ABB RAPID module: P106.mod

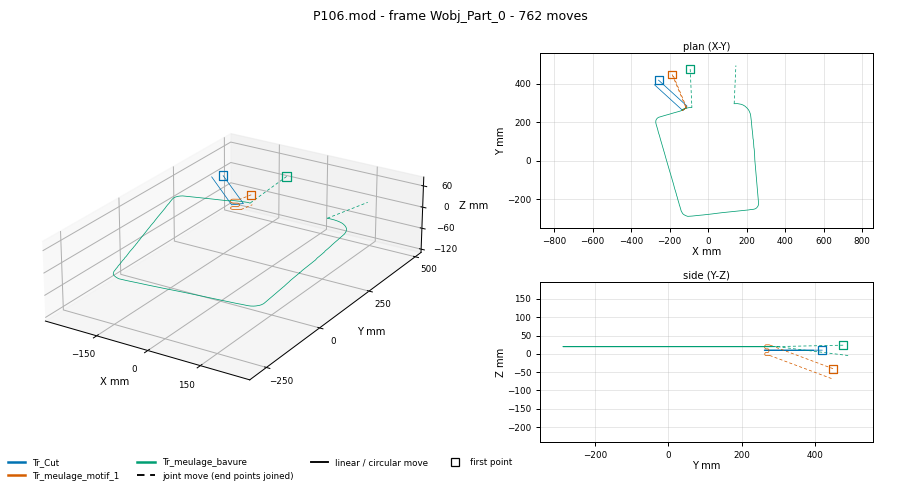
[picture p0: tool path of P106.mod in frame Wobj_Part_0, 762 of 770 moves have a stored position in this frame; points joined in program order, loops and branches not executed]
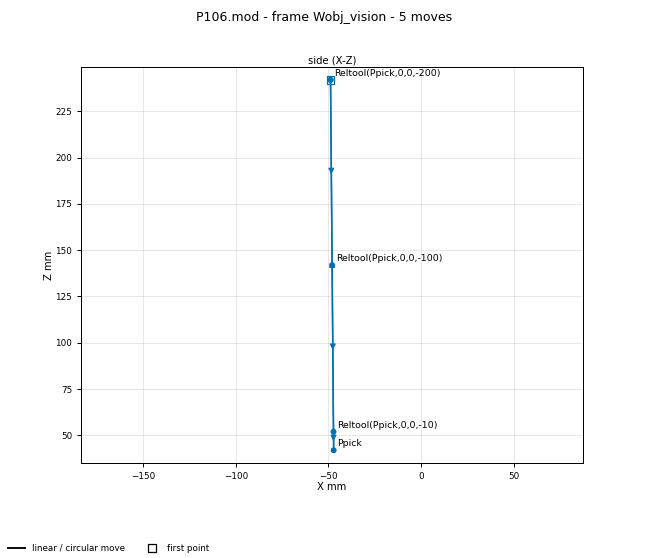
[picture p1: tool path of P106.mod in frame Wobj_vision, 5 of 770 moves have a stored position in this frame; points joined in program order, loops and branches not executed]
MODULE P106
	LOCAL CONST Speeddata vitesse_Tronconnage :=[10, 500, 0, 0];
	LOCAL CONST Robtarget Coupe_0 :=[[-123.979,269.4866875,10.1718701171875],[0.659483403277492,0.659350185940918,-0.255455147334473,-0.255111036220579],[0,0,0,0],[8.999999E+09,8.999999E+09,8.999999E+09,8.999999E+09,8.999999E+09,8.999999E+09]];
	LOCAL CONST Robtarget Tr_meulage_motif_1_App1 :=[[-187.295514074662,449.36288798166,-40.5098213895633],[0.160101054175836,-0.114155213921264,0.569221589744271,-0.798325135114373],[0,0,0,0],[8.999999E+09,8.999999E+09,8.999999E+09,8.999999E+09,8.999999E+09,8.999999E+09]];
	LOCAL CONST Robtarget Tr_meulage_motif_1_App2 :=[[-118.034451875608,283.626825649083,21.4132187938031],[0.160101054175836,-0.114155213921264,0.569221589744271,-0.798325135114373],[0,0,0,0],[8.999999E+09,8.999999E+09,8.999999E+09,8.999999E+09,8.999999E+09,8.999999E+09]];
	LOCAL CONST Robtarget Tr_meulage_motif_1_P0 :=[[-114.3891328125,274.903875,24.672326171875],[0.160101054175836,-0.114155213921264,0.569221589744271,-0.798325135114373],[0,0,0,0],[8.999999E+09,8.999999E+09,8.999999E+09,8.999999E+09,8.999999E+09,8.999999E+09]];
	LOCAL CONST Robtarget Tr_meulage_motif_1_P1 :=[[-115.2604296875,274.413125,24.672283203125],[0.160101054175836,-0.114155213921264,0.569221589744271,-0.798325135114373],[0,0,0,0],[8.999999E+09,8.999999E+09,8.999999E+09,8.999999E+09,8.999999E+09,8.999999E+09]];
	LOCAL CONST Robtarget Tr_meulage_motif_1_P2 :=[[-116.1317265625,273.922375,24.6722421875],[0.160101054175836,-0.114155213921264,0.569221589744271,-0.798325135114373],[0,0,0,0],[8.999999E+09,8.999999E+09,8.999999E+09,8.999999E+09,8.999999E+09,8.999999E+09]];
	LOCAL CONST Robtarget Tr_meulage_motif_1_P3 :=[[-117.0030234375,273.43159375,24.67219921875],[0.160101054175836,-0.114155213921264,0.569221589744271,-0.798325135114373],[0,0,0,0],[8.999999E+09,8.999999E+09,8.999999E+09,8.999999E+09,8.999999E+09,8.999999E+09]];
	LOCAL CONST Robtarget Tr_meulage_motif_1_P4 :=[[-117.8743203125,272.94084375,24.672158203125],[0.160101054175836,-0.114155213921264,0.569221589744271,-0.798325135114373],[0,0,0,0],[8.999999E+09,8.999999E+09,8.999999E+09,8.999999E+09,8.999999E+09,8.999999E+09]];
	LOCAL CONST Robtarget Tr_meulage_motif_1_P5 :=[[-118.745609375,272.45009375,24.672115234375],[0.160101054175836,-0.114155213921264,0.569221589744271,-0.798325135114373],[0,0,0,0],[8.999999E+09,8.999999E+09,8.999999E+09,8.999999E+09,8.999999E+09,8.999999E+09]];
	LOCAL CONST Robtarget Tr_meulage_motif_1_P6 :=[[-119.61690625,271.95934375,24.67207421875],[0.160101054175836,-0.114155213921264,0.569221589744271,-0.798325135114373],[0,0,0,0],[8.999999E+09,8.999999E+09,8.999999E+09,8.999999E+09,8.999999E+09,8.999999E+09]];
	LOCAL CONST Robtarget Tr_meulage_motif_1_P7 :=[[-120.488203125,271.4685625,24.67203125],[0.160101054175836,-0.114155213921264,0.569221589744271,-0.798325135114373],[0,0,0,0],[8.999999E+09,8.999999E+09,8.999999E+09,8.999999E+09,8.999999E+09,8.999999E+09]];
	LOCAL CONST Robtarget Tr_meulage_motif_1_P8 :=[[-121.3595,270.9778125,24.671990234375],[0.160101054175836,-0.114155213921264,0.569221589744271,-0.798325135114373],[0,0,0,0],[8.999999E+09,8.999999E+09,8.999999E+09,8.999999E+09,8.999999E+09,8.999999E+09]];
	LOCAL CONST Robtarget Tr_meulage_motif_1_P9 :=[[-122.230796875,270.4870625,24.671947265625],[0.160101054175836,-0.114155213921264,0.569221589744271,-0.798325135114373],[0,0,0,0],[8.999999E+09,8.999999E+09,8.999999E+09,8.999999E+09,8.999999E+09,8.999999E+09]];
	LOCAL CONST Robtarget Tr_meulage_motif_1_P10 :=[[-123.10209375,269.9963125,24.67190625],[0.160101054175836,-0.114155213921264,0.569221589744271,-0.798325135114373],[0,0,0,0],[8.999999E+09,8.999999E+09,8.999999E+09,8.999999E+09,8.999999E+09,8.999999E+09]];
	LOCAL CONST Robtarget Tr_meulage_motif_1_P11 :=[[-123.973390625,269.50553125,24.671865234375],[0.160101054175836,-0.114155213921264,0.569221589744271,-0.798325135114373],[0,0,0,0],[8.999999E+09,8.999999E+09,8.999999E+09,8.999999E+09,8.999999E+09,8.999999E+09]];
	LOCAL CONST Robtarget Tr_meulage_motif_1_P12 :=[[-124.8446796875,269.01478125,24.671822265625],[0.160101054175836,-0.114155213921264,0.569221589744271,-0.798325135114373],[0,0,0,0],[8.999999E+09,8.999999E+09,8.999999E+09,8.999999E+09,8.999999E+09,8.999999E+09]];
	LOCAL CONST Robtarget Tr_meulage_motif_1_P13 :=[[-125.7159765625,268.52403125,24.67178125],[0.160101054175836,-0.114155213921264,0.569221589744271,-0.798325135114373],[0,0,0,0],[8.999999E+09,8.999999E+09,8.999999E+09,8.999999E+09,8.999999E+09,8.999999E+09]];
	LOCAL CONST Robtarget Tr_meulage_motif_1_P14 :=[[-126.5872734375,268.03325,24.67173828125],[0.160101054175836,-0.114155213921264,0.569221589744271,-0.798325135114373],[0,0,0,0],[8.999999E+09,8.999999E+09,8.999999E+09,8.999999E+09,8.999999E+09,8.999999E+09]];
	LOCAL CONST Robtarget Tr_meulage_motif_1_P15 :=[[-127.4585703125,267.5425,24.671697265625],[0.160101054175836,-0.114155213921264,0.569221589744271,-0.798325135114373],[0,0,0,0],[8.999999E+09,8.999999E+09,8.999999E+09,8.999999E+09,8.999999E+09,8.999999E+09]];
	LOCAL CONST Robtarget Tr_meulage_motif_1_P16 :=[[-128.3298671875,267.05175,24.671654296875],[0.160101054175836,-0.114155213921264,0.569221589744271,-0.798325135114373],[0,0,0,0],[8.999999E+09,8.999999E+09,8.999999E+09,8.999999E+09,8.999999E+09,8.999999E+09]];
	LOCAL CONST Robtarget Tr_meulage_motif_1_P17 :=[[-129.2011640625,266.561,24.67161328125],[0.160101054175836,-0.114155213921264,0.569221589744271,-0.798325135114373],[0,0,0,0],[8.999999E+09,8.999999E+09,8.999999E+09,8.999999E+09,8.999999E+09,8.999999E+09]];
	LOCAL CONST Robtarget Tr_meulage_motif_1_P18 :=[[-130.072453125,266.07021875,24.6715703125],[0.160101054175836,-0.114155213921264,0.569221589744271,-0.798325135114373],[0,0,0,0],[8.999999E+09,8.999999E+09,8.999999E+09,8.999999E+09,8.999999E+09,8.999999E+09]];
	LOCAL CONST Robtarget Tr_meulage_motif_1_P19 :=[[-130.93721875,265.58303125,24.560935546875],[0.160101054175836,-0.114155213921264,0.569221589744271,-0.798325135114373],[0,0,0,0],[8.999999E+09,8.999999E+09,8.999999E+09,8.999999E+09,8.999999E+09,8.999999E+09]];
	LOCAL CONST Robtarget Tr_meulage_motif_1_P20 :=[[-131.761796875,265.118375,24.349708984375],[0.160101054175836,-0.114155213921264,0.569221589744271,-0.798325135114373],[0,0,0,0],[8.999999E+09,8.999999E+09,8.999999E+09,8.999999E+09,8.999999E+09,8.999999E+09]];
	LOCAL CONST Robtarget Tr_meulage_motif_1_P21 :=[[-132.504625,264.69965625,24.077828125],[0.160101054175836,-0.114155213921264,0.569221589744271,-0.798325135114373],[0,0,0,0],[8.999999E+09,8.999999E+09,8.999999E+09,8.999999E+09,8.999999E+09,8.999999E+09]];
	LOCAL CONST Robtarget Tr_meulage_motif_1_P22 :=[[-133.15790625,264.33140625,23.801859375],[0.160101054175836,-0.114155213921264,0.569221589744271,-0.798325135114373],[0,0,0,0],[8.999999E+09,8.999999E+09,8.999999E+09,8.999999E+09,8.999999E+09,8.999999E+09]];
	LOCAL CONST Robtarget Tr_meulage_motif_1_P23 :=[[-134.116953125,263.7905625,23.185689453125],[0.160101054175836,-0.114155213921264,0.569221589744271,-0.798325135114373],[0,0,0,0],[8.999999E+09,8.999999E+09,8.999999E+09,8.999999E+09,8.999999E+09,8.999999E+09]];
	LOCAL CONST Robtarget Tr_meulage_motif_1_P24 :=[[-135.008625,263.28740625,22.337990234375],[0.160101054175836,-0.114155213921264,0.569221589744271,-0.798325135114373],[0,0,0,0],[8.999999E+09,8.999999E+09,8.999999E+09,8.999999E+09,8.999999E+09,8.999999E+09]];
	LOCAL CONST Robtarget Tr_meulage_motif_1_P25 :=[[-135.746671875,262.87059375,21.314080078125],[0.160101054175836,-0.114155213921264,0.569221589744271,-0.798325135114373],[0,0,0,0],[8.999999E+09,8.999999E+09,8.999999E+09,8.999999E+09,8.999999E+09,8.999999E+09]];
	LOCAL CONST Robtarget Tr_meulage_motif_1_P26 :=[[-136.1714375,262.630125,20.197873046875],[0.160101054175836,-0.114155213921264,0.569221589744271,-0.798325135114373],[0,0,0,0],[8.999999E+09,8.999999E+09,8.999999E+09,8.999999E+09,8.999999E+09,8.999999E+09]];
	LOCAL CONST Robtarget Tr_meulage_motif_1_P27 :=[[-136.194671875,262.61628125,19.50190234375],[0.160101054175836,-0.114155213921264,0.569221589744271,-0.798325135114373],[0,0,0,0],[8.999999E+09,8.999999E+09,8.999999E+09,8.999999E+09,8.999999E+09,8.999999E+09]];
	LOCAL CONST Robtarget Tr_meulage_motif_1_P28 :=[[-136.19434375,262.61575,18.840654296875],[0.160101054175836,-0.114155213921264,0.569221589744271,-0.798325135114373],[0,0,0,0],[8.999999E+09,8.999999E+09,8.999999E+09,8.999999E+09,8.999999E+09,8.999999E+09]];
	LOCAL CONST Robtarget Tr_meulage_motif_1_P29 :=[[-136.146203125,262.64215625,18.1795625],[0.160101054175836,-0.114155213921264,0.569221589744271,-0.798325135114373],[0,0,0,0],[8.999999E+09,8.999999E+09,8.999999E+09,8.999999E+09,8.999999E+09,8.999999E+09]];
	LOCAL CONST Robtarget Tr_meulage_motif_1_P30 :=[[-135.7115625,262.88578125,17.077833984375],[0.160101054175836,-0.114155213921264,0.569221589744271,-0.798325135114373],[0,0,0,0],[8.999999E+09,8.999999E+09,8.999999E+09,8.999999E+09,8.999999E+09,8.999999E+09]];
	LOCAL CONST Robtarget Tr_meulage_motif_1_P31 :=[[-134.9646875,263.305375,16.0712451171875],[0.160101054175836,-0.114155213921264,0.569221589744271,-0.798325135114373],[0,0,0,0],[8.999999E+09,8.999999E+09,8.999999E+09,8.999999E+09,8.999999E+09,8.999999E+09]];
	LOCAL CONST Robtarget Tr_meulage_motif_1_P32 :=[[-134.072578125,263.8069375,15.2424130859375],[0.160101054175836,-0.114155213921264,0.569221589744271,-0.798325135114373],[0,0,0,0],[8.999999E+09,8.999999E+09,8.999999E+09,8.999999E+09,8.999999E+09,8.999999E+09]];
	LOCAL CONST Robtarget Tr_meulage_motif_1_P33 :=[[-133.47371875,264.14384375,14.8466923828125],[0.160101054175836,-0.114155213921264,0.569221589744271,-0.798325135114373],[0,0,0,0],[8.999999E+09,8.999999E+09,8.999999E+09,8.999999E+09,8.999999E+09,8.999999E+09]];
	LOCAL CONST Robtarget Tr_meulage_motif_1_P34 :=[[-132.464375,264.7118125,14.3592099609375],[0.160101054175836,-0.114155213921264,0.569221589744271,-0.798325135114373],[0,0,0,0],[8.999999E+09,8.999999E+09,8.999999E+09,8.999999E+09,8.999999E+09,8.999999E+09]];
	LOCAL CONST Robtarget Tr_meulage_motif_1_P35 :=[[-131.72796875,265.1263125,14.0951513671875],[0.160101054175836,-0.114155213921264,0.569221589744271,-0.798325135114373],[0,0,0,0],[8.999999E+09,8.999999E+09,8.999999E+09,8.999999E+09,8.999999E+09,8.999999E+09]];
	LOCAL CONST Robtarget Tr_meulage_motif_1_P36 :=[[-130.915828125,265.58353125,13.8907216796875],[0.160101054175836,-0.114155213921264,0.569221589744271,-0.798325135114373],[0,0,0,0],[8.999999E+09,8.999999E+09,8.999999E+09,8.999999E+09,8.999999E+09,8.999999E+09]];
	LOCAL CONST Robtarget Tr_meulage_motif_1_P37 :=[[-130.0605390625,266.06515625,13.782169921875],[0.160101054175836,-0.114155213921264,0.569221589744271,-0.798325135114373],[0,0,0,0],[8.999999E+09,8.999999E+09,8.999999E+09,8.999999E+09,8.999999E+09,8.999999E+09]];
	LOCAL CONST Robtarget Tr_meulage_motif_1_P38 :=[[-129.195671875,266.5521875,13.6716171875],[0.160101054175836,-0.114155213921264,0.569221589744271,-0.798325135114373],[0,0,0,0],[8.999999E+09,8.999999E+09,8.999999E+09,8.999999E+09,8.999999E+09,8.999999E+09]];
	LOCAL CONST Robtarget Tr_meulage_motif_1_P39 :=[[-128.324375,267.0429375,13.6716591796875],[0.160101054175836,-0.114155213921264,0.569221589744271,-0.798325135114373],[0,0,0,0],[8.999999E+09,8.999999E+09,8.999999E+09,8.999999E+09,8.999999E+09,8.999999E+09]];
	LOCAL CONST Robtarget Tr_meulage_motif_1_P40 :=[[-127.453078125,267.5336875,13.671701171875],[0.160101054175836,-0.114155213921264,0.569221589744271,-0.798325135114373],[0,0,0,0],[8.999999E+09,8.999999E+09,8.999999E+09,8.999999E+09,8.999999E+09,8.999999E+09]];
	LOCAL CONST Robtarget Tr_meulage_motif_1_P41 :=[[-126.58178125,268.02446875,13.6717431640625],[0.160101054175836,-0.114155213921264,0.569221589744271,-0.798325135114373],[0,0,0,0],[8.999999E+09,8.999999E+09,8.999999E+09,8.999999E+09,8.999999E+09,8.999999E+09]];
	LOCAL CONST Robtarget Tr_meulage_motif_1_P42 :=[[-125.710484375,268.51521875,13.67178515625],[0.160101054175836,-0.114155213921264,0.569221589744271,-0.798325135114373],[0,0,0,0],[8.999999E+09,8.999999E+09,8.999999E+09,8.999999E+09,8.999999E+09,8.999999E+09]];
	LOCAL CONST Robtarget Tr_meulage_motif_1_P43 :=[[-124.8391875,269.00596875,13.6718271484375],[0.160101054175836,-0.114155213921264,0.569221589744271,-0.798325135114373],[0,0,0,0],[8.999999E+09,8.999999E+09,8.999999E+09,8.999999E+09,8.999999E+09,8.999999E+09]];
	LOCAL CONST Robtarget Tr_meulage_motif_1_P44 :=[[-123.9678984375,269.49671875,13.671869140625],[0.160101054175836,-0.114155213921264,0.569221589744271,-0.798325135114373],[0,0,0,0],[8.999999E+09,8.999999E+09,8.999999E+09,8.999999E+09,8.999999E+09,8.999999E+09]];
	LOCAL CONST Robtarget Tr_meulage_motif_1_P45 :=[[-123.0966015625,269.9875,13.6719111328125],[0.160101054175836,-0.114155213921264,0.569221589744271,-0.798325135114373],[0,0,0,0],[8.999999E+09,8.999999E+09,8.999999E+09,8.999999E+09,8.999999E+09,8.999999E+09]];
	LOCAL CONST Robtarget Tr_meulage_motif_1_P46 :=[[-122.2253046875,270.47825,13.671953125],[0.160101054175836,-0.114155213921264,0.569221589744271,-0.798325135114373],[0,0,0,0],[8.999999E+09,8.999999E+09,8.999999E+09,8.999999E+09,8.999999E+09,8.999999E+09]];
	LOCAL CONST Robtarget Tr_meulage_motif_1_P47 :=[[-121.3540078125,270.969,13.6719951171875],[0.160101054175836,-0.114155213921264,0.569221589744271,-0.798325135114373],[0,0,0,0],[8.999999E+09,8.999999E+09,8.999999E+09,8.999999E+09,8.999999E+09,8.999999E+09]];
	LOCAL CONST Robtarget Tr_meulage_motif_1_P48 :=[[-120.4827109375,271.45975,13.672037109375],[0.160101054175836,-0.114155213921264,0.569221589744271,-0.798325135114373],[0,0,0,0],[8.999999E+09,8.999999E+09,8.999999E+09,8.999999E+09,8.999999E+09,8.999999E+09]];
	LOCAL CONST Robtarget Tr_meulage_motif_1_P49 :=[[-119.61784375,271.94678125,13.5614853515625],[0.160101054175836,-0.114155213921264,0.569221589744271,-0.798325135114373],[0,0,0,0],[8.999999E+09,8.999999E+09,8.999999E+09,8.999999E+09,8.999999E+09,8.999999E+09]];
	LOCAL CONST Robtarget Tr_meulage_motif_1_P50 :=[[-118.7930546875,272.411125,13.3503369140625],[0.160101054175836,-0.114155213921264,0.569221589744271,-0.798325135114373],[0,0,0,0],[8.999999E+09,8.999999E+09,8.999999E+09,8.999999E+09,8.999999E+09,8.999999E+09]];
	LOCAL CONST Robtarget Tr_meulage_motif_1_P51 :=[[-118.049953125,272.829375,13.078529296875],[0.160101054175836,-0.114155213921264,0.569221589744271,-0.798325135114373],[0,0,0,0],[8.999999E+09,8.999999E+09,8.999999E+09,8.999999E+09,8.999999E+09,8.999999E+09]];
	LOCAL CONST Robtarget Tr_meulage_motif_1_P52 :=[[-117.4298671875,273.1783125,12.7744033203125],[0.160101054175836,-0.114155213921264,0.569221589744271,-0.798325135114373],[0,0,0,0],[8.999999E+09,8.999999E+09,8.999999E+09,8.999999E+09,8.999999E+09,8.999999E+09]];
	LOCAL CONST Robtarget Tr_meulage_motif_1_P53 :=[[-116.5282109375,273.6854375,12.111916015625],[0.160101054175836,-0.114155213921264,0.569221589744271,-0.798325135114373],[0,0,0,0],[8.999999E+09,8.999999E+09,8.999999E+09,8.999999E+09,8.999999E+09,8.999999E+09]];
	LOCAL CONST Robtarget Tr_meulage_motif_1_P54 :=[[-115.74190625,274.127375,11.2100166015625],[0.160101054175836,-0.114155213921264,0.569221589744271,-0.798325135114373],[0,0,0,0],[8.999999E+09,8.999999E+09,8.999999E+09,8.999999E+09,8.999999E+09,8.999999E+09]];
	LOCAL CONST Robtarget Tr_meulage_motif_1_P55 :=[[-115.275265625,274.3890625,10.1640078125],[0.160101054175836,-0.114155213921264,0.569221589744271,-0.798325135114373],[0,0,0,0],[8.999999E+09,8.999999E+09,8.999999E+09,8.999999E+09,8.999999E+09,8.999999E+09]];
	LOCAL CONST Robtarget Tr_meulage_motif_1_P56 :=[[-115.113921875,274.4791875,9.470796875],[0.160101054175836,-0.114155213921264,0.569221589744271,-0.798325135114373],[0,0,0,0],[8.999999E+09,8.999999E+09,8.999999E+09,8.999999E+09,8.999999E+09,8.999999E+09]];
	LOCAL CONST Robtarget Tr_meulage_motif_1_P57 :=[[-115.0579140625,274.50990625,8.7007998046875],[0.160101054175836,-0.114155213921264,0.569221589744271,-0.798325135114373],[0,0,0,0],[8.999999E+09,8.999999E+09,8.999999E+09,8.999999E+09,8.999999E+09,8.999999E+09]];
	LOCAL CONST Robtarget Tr_meulage_motif_1_P58 :=[[-115.1158515625,274.4764375,7.9309228515625],[0.160101054175836,-0.114155213921264,0.569221589744271,-0.798325135114373],[0,0,0,0],[8.999999E+09,8.999999E+09,8.999999E+09,8.999999E+09,8.999999E+09,8.999999E+09]];
	LOCAL CONST Robtarget Tr_meulage_motif_1_P59 :=[[-115.480890625,274.269625,6.82265576171875],[0.160101054175836,-0.114155213921264,0.569221589744271,-0.798325135114373],[0,0,0,0],[8.999999E+09,8.999999E+09,8.999999E+09,8.999999E+09,8.999999E+09,8.999999E+09]];
	LOCAL CONST Robtarget Tr_meulage_motif_1_P60 :=[[-115.8415859375,274.06584375,6.236951171875],[0.160101054175836,-0.114155213921264,0.569221589744271,-0.798325135114373],[0,0,0,0],[8.999999E+09,8.999999E+09,8.999999E+09,8.999999E+09,8.999999E+09,8.999999E+09]];
	LOCAL CONST Robtarget Tr_meulage_motif_1_P61 :=[[-116.6140859375,273.62975,5.3497890625],[0.160101054175836,-0.114155213921264,0.569221589744271,-0.798325135114373],[0,0,0,0],[8.999999E+09,8.999999E+09,8.999999E+09,8.999999E+09,8.999999E+09,8.999999E+09]];
	LOCAL CONST Robtarget Tr_meulage_motif_1_P62 :=[[-117.1241875,273.342,4.9354521484375],[0.160101054175836,-0.114155213921264,0.569221589744271,-0.798325135114373],[0,0,0,0],[8.999999E+09,8.999999E+09,8.999999E+09,8.999999E+09,8.999999E+09,8.999999E+09]];
	LOCAL CONST Robtarget Tr_meulage_motif_1_P63 :=[[-118.0979453125,272.7929375,4.39131201171875],[0.160101054175836,-0.114155213921264,0.569221589744271,-0.798325135114373],[0,0,0,0],[8.999999E+09,8.999999E+09,8.999999E+09,8.999999E+09,8.999999E+09,8.999999E+09]];
	LOCAL CONST Robtarget Tr_meulage_motif_1_P64 :=[[-118.8171328125,272.38753125,4.09577734375],[0.160101054175836,-0.114155213921264,0.569221589744271,-0.798325135114373],[0,0,0,0],[8.999999E+09,8.999999E+09,8.999999E+09,8.999999E+09,8.999999E+09,8.999999E+09]];
	LOCAL CONST Robtarget Tr_meulage_motif_1_P65 :=[[-119.629078125,271.93,3.89126977539062],[0.160101054175836,-0.114155213921264,0.569221589744271,-0.798325135114373],[0,0,0,0],[8.999999E+09,8.999999E+09,8.999999E+09,8.999999E+09,8.999999E+09,8.999999E+09]];
	LOCAL CONST Robtarget Tr_meulage_motif_1_P66 :=[[-120.4842578125,271.4481875,3.782634765625],[0.160101054175836,-0.114155213921264,0.569221589744271,-0.798325135114373],[0,0,0,0],[8.999999E+09,8.999999E+09,8.999999E+09,8.999999E+09,8.999999E+09,8.999999E+09]];
	LOCAL CONST Robtarget Tr_meulage_motif_1_P67 :=[[-121.349015625,270.961,3.67199951171875],[0.160101054175836,-0.114155213921264,0.569221589744271,-0.798325135114373],[0,0,0,0],[8.999999E+09,8.999999E+09,8.999999E+09,8.999999E+09,8.999999E+09,8.999999E+09]];
	LOCAL CONST Robtarget Tr_meulage_motif_1_P68 :=[[-122.2203125,270.47025,3.67195751953125],[0.160101054175836,-0.114155213921264,0.569221589744271,-0.798325135114373],[0,0,0,0],[8.999999E+09,8.999999E+09,8.999999E+09,8.999999E+09,8.999999E+09,8.999999E+09]];
	LOCAL CONST Robtarget Tr_meulage_motif_1_P69 :=[[-123.091609375,269.97946875,3.67191552734375],[0.160101054175836,-0.114155213921264,0.569221589744271,-0.798325135114373],[0,0,0,0],[8.999999E+09,8.999999E+09,8.999999E+09,8.999999E+09,8.999999E+09,8.999999E+09]];
	LOCAL CONST Robtarget Tr_meulage_motif_1_P70 :=[[-123.96290625,269.48871875,3.67187353515625],[0.160101054175836,-0.114155213921264,0.569221589744271,-0.798325135114373],[0,0,0,0],[8.999999E+09,8.999999E+09,8.999999E+09,8.999999E+09,8.999999E+09,8.999999E+09]];
	LOCAL CONST Robtarget Tr_meulage_motif_1_P71 :=[[-124.8341953125,268.99796875,3.67183178710938],[0.160101054175836,-0.114155213921264,0.569221589744271,-0.798325135114373],[0,0,0,0],[8.999999E+09,8.999999E+09,8.999999E+09,8.999999E+09,8.999999E+09,8.999999E+09]];
	LOCAL CONST Robtarget Tr_meulage_motif_1_P72 :=[[-125.7054921875,268.50721875,3.67178979492187],[0.160101054175836,-0.114155213921264,0.569221589744271,-0.798325135114373],[0,0,0,0],[8.999999E+09,8.999999E+09,8.999999E+09,8.999999E+09,8.999999E+09,8.999999E+09]];
	LOCAL CONST Robtarget Tr_meulage_motif_1_P73 :=[[-126.5767890625,268.0164375,3.67174780273438],[0.160101054175836,-0.114155213921264,0.569221589744271,-0.798325135114373],[0,0,0,0],[8.999999E+09,8.999999E+09,8.999999E+09,8.999999E+09,8.999999E+09,8.999999E+09]];
	LOCAL CONST Robtarget Tr_meulage_motif_1_P74 :=[[-127.4480859375,267.5256875,3.67170581054688],[0.160101054175836,-0.114155213921264,0.569221589744271,-0.798325135114373],[0,0,0,0],[8.999999E+09,8.999999E+09,8.999999E+09,8.999999E+09,8.999999E+09,8.999999E+09]];
	LOCAL CONST Robtarget Tr_meulage_motif_1_P75 :=[[-128.3193828125,267.0349375,3.67166381835938],[0.160101054175836,-0.114155213921264,0.569221589744271,-0.798325135114373],[0,0,0,0],[8.999999E+09,8.999999E+09,8.999999E+09,8.999999E+09,8.999999E+09,8.999999E+09]];
	LOCAL CONST Robtarget Tr_meulage_motif_1_P76 :=[[-129.1906796875,266.54415625,3.67162182617187],[0.160101054175836,-0.114155213921264,0.569221589744271,-0.798325135114373],[0,0,0,0],[8.999999E+09,8.999999E+09,8.999999E+09,8.999999E+09,8.999999E+09,8.999999E+09]];
	LOCAL CONST Robtarget Tr_meulage_motif_1_P77 :=[[-130.0619765625,266.05340625,3.671580078125],[0.160101054175836,-0.114155213921264,0.569221589744271,-0.798325135114373],[0,0,0,0],[8.999999E+09,8.999999E+09,8.999999E+09,8.999999E+09,8.999999E+09,8.999999E+09]];
	LOCAL CONST Robtarget Tr_meulage_motif_1_P78 :=[[-130.926734375,265.56621875,3.56094458007813],[0.160101054175836,-0.114155213921264,0.569221589744271,-0.798325135114373],[0,0,0,0],[8.999999E+09,8.999999E+09,8.999999E+09,8.999999E+09,8.999999E+09,8.999999E+09]];
	LOCAL CONST Robtarget Tr_meulage_motif_1_P79 :=[[-131.7513125,265.10153125,3.34971752929688],[0.160101054175836,-0.114155213921264,0.569221589744271,-0.798325135114373],[0,0,0,0],[8.999999E+09,8.999999E+09,8.999999E+09,8.999999E+09,8.999999E+09,8.999999E+09]];
	LOCAL CONST Robtarget Tr_meulage_motif_1_P80 :=[[-132.494140625,264.68284375,3.07783813476563],[0.160101054175836,-0.114155213921264,0.569221589744271,-0.798325135114373],[0,0,0,0],[8.999999E+09,8.999999E+09,8.999999E+09,8.999999E+09,8.999999E+09,8.999999E+09]];
	LOCAL CONST Robtarget Tr_meulage_motif_1_P81 :=[[-133.147421875,264.31459375,2.80186938476563],[0.160101054175836,-0.114155213921264,0.569221589744271,-0.798325135114373],[0,0,0,0],[8.999999E+09,8.999999E+09,8.999999E+09,8.999999E+09,8.999999E+09,8.999999E+09]];
	LOCAL CONST Robtarget Tr_meulage_motif_1_P82 :=[[-134.10646875,263.77375,2.18569848632813],[0.160101054175836,-0.114155213921264,0.569221589744271,-0.798325135114373],[0,0,0,0],[8.999999E+09,8.999999E+09,8.999999E+09,8.999999E+09,8.999999E+09,8.999999E+09]];
	LOCAL CONST Robtarget Tr_meulage_motif_1_P83 :=[[-134.939609375,263.3035,1.29168994140625],[0.160101054175836,-0.114155213921264,0.569221589744271,-0.798325135114373],[0,0,0,0],[8.999999E+09,8.999999E+09,8.999999E+09,8.999999E+09,8.999999E+09,8.999999E+09]];
	LOCAL CONST Robtarget Tr_meulage_motif_1_P84 :=[[-135.469796875,263.0036875,0.205664825439453],[0.160101054175836,-0.114155213921264,0.569221589744271,-0.798325135114373],[0,0,0,0],[8.999999E+09,8.999999E+09,8.999999E+09,8.999999E+09,8.999999E+09,8.999999E+09]];
	LOCAL CONST Robtarget Tr_meulage_motif_1_P85 :=[[-135.616828125,262.9198125,-0.778716857910156],[0.160101054175836,-0.114155213921264,0.569221589744271,-0.798325135114373],[0,0,0,0],[8.999999E+09,8.999999E+09,8.999999E+09,8.999999E+09,8.999999E+09,8.999999E+09]];
	LOCAL CONST Robtarget Tr_meulage_motif_1_P86 :=[[-135.502171875,262.9841875,-0.983367492675781],[0.160101054175836,-0.114155213921264,0.569221589744271,-0.798325135114373],[0,0,0,0],[8.999999E+09,8.999999E+09,8.999999E+09,8.999999E+09,8.999999E+09,8.999999E+09]];
	LOCAL CONST Robtarget Tr_meulage_motif_1_P87 :=[[-135.3943125,263.04415625,-1.70976818847656],[0.160101054175836,-0.114155213921264,0.569221589744271,-0.798325135114373],[0,0,0,0],[8.999999E+09,8.999999E+09,8.999999E+09,8.999999E+09,8.999999E+09,8.999999E+09]];
	LOCAL CONST Robtarget Tr_meulage_motif_1_P88 :=[[-134.797875,263.3790625,-2.64664526367187],[0.160101054175836,-0.114155213921264,0.569221589744271,-0.798325135114373],[0,0,0,0],[8.999999E+09,8.999999E+09,8.999999E+09,8.999999E+09,8.999999E+09,8.999999E+09]];
	LOCAL CONST Robtarget Tr_meulage_motif_1_P89 :=[[-134.311796875,263.65234375,-3.11043432617187],[0.160101054175836,-0.114155213921264,0.569221589744271,-0.798325135114373],[0,0,0,0],[8.999999E+09,8.999999E+09,8.999999E+09,8.999999E+09,8.999999E+09,8.999999E+09]];
	LOCAL CONST Robtarget Tr_meulage_motif_1_P90 :=[[-133.3266875,264.20665625,-3.64082421875],[0.160101054175836,-0.114155213921264,0.569221589744271,-0.798325135114373],[0,0,0,0],[8.999999E+09,8.999999E+09,8.999999E+09,8.999999E+09,8.999999E+09,8.999999E+09]];
	LOCAL CONST Robtarget Tr_meulage_motif_1_P91 :=[[-132.59028125,264.621125,-3.90488232421875],[0.160101054175836,-0.114155213921264,0.569221589744271,-0.798325135114373],[0,0,0,0],[8.999999E+09,8.999999E+09,8.999999E+09,8.999999E+09,8.999999E+09,8.999999E+09]];
	LOCAL CONST Robtarget Tr_meulage_motif_1_P92 :=[[-131.778140625,265.078375,-4.10931201171875],[0.160101054175836,-0.114155213921264,0.569221589744271,-0.798325135114373],[0,0,0,0],[8.999999E+09,8.999999E+09,8.999999E+09,8.999999E+09,8.999999E+09,8.999999E+09]];
	LOCAL CONST Robtarget Tr_meulage_motif_1_P93 :=[[-130.9228515625,265.56,-4.2178642578125],[0.160101054175836,-0.114155213921264,0.569221589744271,-0.798325135114373],[0,0,0,0],[8.999999E+09,8.999999E+09,8.999999E+09,8.999999E+09,8.999999E+09,8.999999E+09]];
	LOCAL CONST Robtarget Tr_meulage_motif_1_P94 :=[[-130.0579765625,266.047,-4.32841650390625],[0.160101054175836,-0.114155213921264,0.569221589744271,-0.798325135114373],[0,0,0,0],[8.999999E+09,8.999999E+09,8.999999E+09,8.999999E+09,8.999999E+09,8.999999E+09]];
	LOCAL CONST Robtarget Tr_meulage_motif_1_P95 :=[[-129.1866875,266.53775,-4.32837451171875],[0.160101054175836,-0.114155213921264,0.569221589744271,-0.798325135114373],[0,0,0,0],[8.999999E+09,8.999999E+09,8.999999E+09,8.999999E+09,8.999999E+09,8.999999E+09]];
	LOCAL CONST Robtarget Tr_meulage_motif_1_P96 :=[[-128.315390625,267.02853125,-4.32833251953125],[0.160101054175836,-0.114155213921264,0.569221589744271,-0.798325135114373],[0,0,0,0],[8.999999E+09,8.999999E+09,8.999999E+09,8.999999E+09,8.999999E+09,8.999999E+09]];
	LOCAL CONST Robtarget Tr_meulage_motif_1_P97 :=[[-127.44409375,267.51928125,-4.32829052734375],[0.160101054175836,-0.114155213921264,0.569221589744271,-0.798325135114373],[0,0,0,0],[8.999999E+09,8.999999E+09,8.999999E+09,8.999999E+09,8.999999E+09,8.999999E+09]];
	LOCAL CONST Robtarget Tr_meulage_motif_1_P98 :=[[-126.572796875,268.01003125,-4.32824853515625],[0.160101054175836,-0.114155213921264,0.569221589744271,-0.798325135114373],[0,0,0,0],[8.999999E+09,8.999999E+09,8.999999E+09,8.999999E+09,8.999999E+09,8.999999E+09]];
	LOCAL CONST Robtarget Tr_meulage_motif_1_P99 :=[[-125.7015,268.5008125,-4.32820654296875],[0.160101054175836,-0.114155213921264,0.569221589744271,-0.798325135114373],[0,0,0,0],[8.999999E+09,8.999999E+09,8.999999E+09,8.999999E+09,8.999999E+09,8.999999E+09]];
	LOCAL CONST Robtarget Tr_meulage_motif_1_P100 :=[[-124.830203125,268.9915625,-4.32816455078125],[0.160101054175836,-0.114155213921264,0.569221589744271,-0.798325135114373],[0,0,0,0],[8.999999E+09,8.999999E+09,8.999999E+09,8.999999E+09,8.999999E+09,8.999999E+09]];
	LOCAL CONST Robtarget Tr_meulage_motif_1_P101 :=[[-123.95890625,269.4823125,-4.328123046875],[0.160101054175836,-0.114155213921264,0.569221589744271,-0.798325135114373],[0,0,0,0],[8.999999E+09,8.999999E+09,8.999999E+09,8.999999E+09,8.999999E+09,8.999999E+09]];
	LOCAL CONST Robtarget Tr_meulage_motif_1_P102 :=[[-123.0876171875,269.9730625,-4.3280810546875],[0.160101054175836,-0.114155213921264,0.569221589744271,-0.798325135114373],[0,0,0,0],[8.999999E+09,8.999999E+09,8.999999E+09,8.999999E+09,8.999999E+09,8.999999E+09]];
	LOCAL CONST Robtarget Tr_meulage_motif_1_P103 :=[[-122.2163203125,270.46384375,-4.3280390625],[0.160101054175836,-0.114155213921264,0.569221589744271,-0.798325135114373],[0,0,0,0],[8.999999E+09,8.999999E+09,8.999999E+09,8.999999E+09,8.999999E+09,8.999999E+09]];
	LOCAL CONST Robtarget Tr_meulage_motif_1_P104 :=[[-121.3450234375,270.95459375,-4.3279970703125],[0.160101054175836,-0.114155213921264,0.569221589744271,-0.798325135114373],[0,0,0,0],[8.999999E+09,8.999999E+09,8.999999E+09,8.999999E+09,8.999999E+09,8.999999E+09]];
	LOCAL CONST Robtarget Tr_meulage_motif_1_P105 :=[[-120.4737265625,271.44534375,-4.327955078125],[0.160101054175836,-0.114155213921264,0.569221589744271,-0.798325135114373],[0,0,0,0],[8.999999E+09,8.999999E+09,8.999999E+09,8.999999E+09,8.999999E+09,8.999999E+09]];
	LOCAL CONST Robtarget Tr_meulage_motif_1_P106 :=[[-119.6024296875,271.93609375,-4.3279130859375],[0.160101054175836,-0.114155213921264,0.569221589744271,-0.798325135114373],[0,0,0,0],[8.999999E+09,8.999999E+09,8.999999E+09,8.999999E+09,8.999999E+09,8.999999E+09]];
	LOCAL CONST Robtarget Tr_meulage_motif_1_P107 :=[[-118.7311328125,272.426875,-4.32787109375],[0.160101054175836,-0.114155213921264,0.569221589744271,-0.798325135114373],[0,0,0,0],[8.999999E+09,8.999999E+09,8.999999E+09,8.999999E+09,8.999999E+09,8.999999E+09]];
	LOCAL CONST Robtarget Tr_meulage_motif_1_P108 :=[[-117.85984375,272.917625,-4.3278291015625],[0.160101054175836,-0.114155213921264,0.569221589744271,-0.798325135114373],[0,0,0,0],[8.999999E+09,8.999999E+09,8.999999E+09,8.999999E+09,8.999999E+09,8.999999E+09]];
	LOCAL CONST Robtarget Tr_meulage_motif_1_P109 :=[[-116.988546875,273.408375,-4.327787109375],[0.160101054175836,-0.114155213921264,0.569221589744271,-0.798325135114373],[0,0,0,0],[8.999999E+09,8.999999E+09,8.999999E+09,8.999999E+09,8.999999E+09,8.999999E+09]];
	LOCAL CONST Robtarget Tr_meulage_motif_1_P110 :=[[-116.11725,273.899125,-4.3277451171875],[0.160101054175836,-0.114155213921264,0.569221589744271,-0.798325135114373],[0,0,0,0],[8.999999E+09,8.999999E+09,8.999999E+09,8.999999E+09,8.999999E+09,8.999999E+09]];
	LOCAL CONST Robtarget Tr_meulage_motif_1_P111 :=[[-115.245953125,274.38990625,-4.327703125],[0.160101054175836,-0.114155213921264,0.569221589744271,-0.798325135114373],[0,0,0,0],[8.999999E+09,8.999999E+09,8.999999E+09,8.999999E+09,8.999999E+09,8.999999E+09]];
	LOCAL CONST Robtarget Tr_meulage_motif_1_P112 :=[[-114.37465625,274.88065625,-4.3276611328125],[0.160101054175836,-0.114155213921264,0.569221589744271,-0.798325135114373],[0,0,0,0],[8.999999E+09,8.999999E+09,8.999999E+09,8.999999E+09,8.999999E+09,8.999999E+09]];
	LOCAL CONST Robtarget Tr_meulage_motif_1_P113 :=[[-113.503359375,275.37140625,-4.32761962890625],[0.160101054175836,-0.114155213921264,0.569221589744271,-0.798325135114373],[0,0,0,0],[8.999999E+09,8.999999E+09,8.999999E+09,8.999999E+09,8.999999E+09,8.999999E+09]];
	LOCAL CONST Robtarget Tr_meulage_motif_1_P114 :=[[-112.6320625,275.8621875,-4.32757763671875],[0.160101054175836,-0.114155213921264,0.569221589744271,-0.798325135114373],[0,0,0,0],[8.999999E+09,8.999999E+09,8.999999E+09,8.999999E+09,8.999999E+09,8.999999E+09]];
	LOCAL CONST Robtarget Tr_meulage_motif_1_P115 :=[[-111.7607734375,276.3529375,-4.32753564453125],[0.160101054175836,-0.114155213921264,0.569221589744271,-0.798325135114373],[0,0,0,0],[8.999999E+09,8.999999E+09,8.999999E+09,8.999999E+09,8.999999E+09,8.999999E+09]];
	LOCAL CONST Robtarget Tr_meulage_motif_1_degg1 :=[[-115.406092500608,285.075888149083,-7.58664302260317],[0.160101054175836,-0.114155213921264,0.569221589744271,-0.798325135114373],[0,0,0,0],[8.999999E+09,8.999999E+09,8.999999E+09,8.999999E+09,8.999999E+09,8.999999E+09]];
	LOCAL CONST Robtarget Tr_meulage_motif_1_degg2 :=[[-184.667154699662,450.81195048166,-69.5096832059696],[0.160101054175836,-0.114155213921264,0.569221589744271,-0.798325135114373],[0,0,0,0],[8.999999E+09,8.999999E+09,8.999999E+09,8.999999E+09,8.999999E+09,8.999999E+09]];
	LOCAL CONST Robtarget Tr_meulage_bavure_App1 :=[[-93.3172790242901,477.040233950797,23.6650555157886],[0.0151955200750049,-0.0155153358033377,0.714263195988972,-0.699540175672691],[0,0,0,0],[8.999999E+09,8.999999E+09,8.999999E+09,8.999999E+09,8.999999E+09,8.999999E+09]];
	LOCAL CONST Robtarget Tr_meulage_bavure_App2 :=[[-85.0685424668395,287.26061951004,19.7082527757894],[0.0151955200750049,-0.0155153358033377,0.714263195988972,-0.699540175672691],[0,0,0,0],[8.999999E+09,8.999999E+09,8.999999E+09,8.999999E+09,8.999999E+09,8.999999E+09]];
	LOCAL CONST Robtarget Tr_meulage_bavure_P0 :=[[-84.6343984375,277.27221875,19.5],[0.0151955200750049,-0.0155153358033377,0.714263195988972,-0.699540175672691],[0,0,0,0],[8.999999E+09,8.999999E+09,8.999999E+09,8.999999E+09,8.999999E+09,8.999999E+09]];
	LOCAL CONST Robtarget Tr_meulage_bavure_P1 :=[[-85.6453515625,277.53284375,19.5],[0.0158206762787373,-0.0161539658647217,0.714255890083302,-0.699519320012131],[0,0,0,0],[8.999999E+09,8.999999E+09,8.999999E+09,8.999999E+09,8.999999E+09,8.999999E+09]];
	LOCAL CONST Robtarget Tr_meulage_bavure_P2 :=[[-88.073609375,278.0285625,19.5],[0.0176886598730735,-0.0180613966765676,0.714212041687733,-0.699472699088553],[0,0,0,0],[8.999999E+09,8.999999E+09,8.999999E+09,8.999999E+09,8.999999E+09,8.999999E+09]];
	LOCAL CONST Robtarget Tr_meulage_bavure_P3 :=[[-91.6300625,278.3053125,19.5],[0.0207426241435952,-0.0211805767672185,0.714140594494554,-0.699374247457261],[0,0,0,0],[8.999999E+09,8.999999E+09,8.999999E+09,8.999999E+09,8.999999E+09,8.999999E+09]];
	LOCAL CONST Robtarget Tr_meulage_bavure_P4 :=[[-91.9578515625,278.3040625,19.5],[0.0249264353407532,-0.0254540680694285,0.714019535108151,-0.699218754556727],[0,0,0,0],[8.999999E+09,8.999999E+09,8.999999E+09,8.999999E+09,8.999999E+09,8.999999E+09]];
	LOCAL CONST Robtarget Tr_meulage_bavure_P5 :=[[-92.130796875,278.2993125,19.5],[0.030127768935588,-0.0307674329619474,0.713832296920205,-0.698991512453134],[0,0,0,0],[8.999999E+09,8.999999E+09,8.999999E+09,8.999999E+09,8.999999E+09,8.999999E+09]];
	LOCAL CONST Robtarget Tr_meulage_bavure_P6 :=[[-92.44025,278.27190625,19.5],[0.0362546568906457,-0.0370277001867813,0.713566120277983,-0.698668692059438],[0,0,0,0],[8.999999E+09,8.999999E+09,8.999999E+09,8.999999E+09,8.999999E+09,8.999999E+09]];
	LOCAL CONST Robtarget Tr_meulage_bavure_P7 :=[[-95.7801796875,277.864375,19.5],[0.0431915252982847,-0.0441163098439704,0.713193375957515,-0.69824311800295],[0,0,0,0],[8.999999E+09,8.999999E+09,8.999999E+09,8.999999E+09,8.999999E+09,8.999999E+09]];
	LOCAL CONST Robtarget Tr_meulage_bavure_P8 :=[[-99.2706640625,277.17515625,19.5],[0.0508095462580043,-0.0519026892623459,0.712704481861975,-0.697693931742455],[0,0,0,0],[8.999999E+09,8.999999E+09,8.999999E+09,8.999999E+09,8.999999E+09,8.999999E+09]];
	LOCAL CONST Robtarget Tr_meulage_bavure_P9 :=[[-102.208890625,276.51165625,19.5],[0.0589863673229863,-0.06026222118999,0.712085915426012,-0.697009843703218],[0,0,0,0],[8.999999E+09,8.999999E+09,8.999999E+09,8.999999E+09,8.999999E+09,8.999999E+09]];
	LOCAL CONST Robtarget Tr_meulage_bavure_P10 :=[[-104.97009375,275.98846875,19.5],[0.0676120560400716,-0.0690827233947068,0.711326296199233,-0.696183228426171],[0,0,0,0],[8.999999E+09,8.999999E+09,8.999999E+09,8.999999E+09,8.999999E+09,8.999999E+09]];
	LOCAL CONST Robtarget Tr_meulage_bavure_P11 :=[[-107.1077578125,275.53821875,19.5],[0.0765702546263699,-0.0782467761945103,0.710426085919104,-0.695204440842607],[0,0,0,0],[8.999999E+09,8.999999E+09,8.999999E+09,8.999999E+09,8.999999E+09,8.999999E+09]];
	LOCAL CONST Robtarget Tr_meulage_bavure_P12 :=[[-109.0425390625,275.0786875,19.5],[0.0857454442227747,-0.0876355069848646,0.709379965946049,-0.694080543326873],[0,0,0,0],[8.999999E+09,8.999999E+09,8.999999E+09,8.999999E+09,8.999999E+09,8.999999E+09]];
	LOCAL CONST Robtarget Tr_meulage_bavure_P13 :=[[-111.625484375,274.48096875,19.5],[0.0950145148772524,-0.0971250552864648,0.7082018155395,-0.692812495603823],[0,0,0,0],[8.999999E+09,8.999999E+09,8.999999E+09,8.999999E+09,8.999999E+09,8.999999E+09]];
	LOCAL CONST Robtarget Tr_meulage_bavure_P14 :=[[-116.3591328125,273.19275,19.5],[0.10425150879754,-0.106587082953937,0.706905496063988,-0.691415530846201],[0,0,0,0],[8.999999E+09,8.999999E+09,8.999999E+09,8.999999E+09,8.999999E+09,8.999999E+09]];
	LOCAL CONST Robtarget Tr_meulage_bavure_P15 :=[[-119.39590625,272.391,19.5],[0.113310966428969,-0.115875110844145,0.70552080380574,-0.689908674370089],[0,0,0,0],[8.999999E+09,8.999999E+09,8.999999E+09,8.999999E+09,8.999999E+09,8.999999E+09]];
	LOCAL CONST Robtarget Tr_meulage_bavure_P16 :=[[-120.538359375,272.08415625,19.5],[0.122055376314245,-0.124844213990626,0.70406527669606,-0.688337485174788],[0,0,0,0],[8.999999E+09,8.999999E+09,8.999999E+09,8.999999E+09,8.999999E+09,8.999999E+09]];
	LOCAL CONST Robtarget Tr_meulage_bavure_P17 :=[[-125.99746875,270.4395625,19.5],[0.130309780759485,-0.133317886714664,0.702591836779638,-0.686738970068661],[0,0,0,0],[8.999999E+09,8.999999E+09,8.999999E+09,8.999999E+09,8.999999E+09,8.999999E+09]];
	LOCAL CONST Robtarget Tr_meulage_bavure_P18 :=[[-127.7929375,269.900375,19.5],[0.137924746777725,-0.141143841092413,0.701150496102952,-0.685159223949123],[0,0,0,0],[8.999999E+09,8.999999E+09,8.999999E+09,8.999999E+09,8.999999E+09,8.999999E+09]];
	LOCAL CONST Robtarget Tr_meulage_bavure_P19 :=[[-129.1219140625,269.4395625,19.5],[0.144724386283821,-0.148136167501402,0.69978849943801,-0.683671400562483],[0,0,0,0],[8.999999E+09,8.999999E+09,8.999999E+09,8.999999E+09,8.999999E+09,8.999999E+09]];
	LOCAL CONST Robtarget Tr_meulage_bavure_P20 :=[[-130.974734375,268.56940625,19.5],[0.150574584511112,-0.15416287139529,0.698575112394482,-0.682315114830019],[0,0,0,0],[8.999999E+09,8.999999E+09,8.999999E+09,8.999999E+09,8.999999E+09,8.999999E+09]];
	LOCAL CONST Robtarget Tr_meulage_bavure_P21 :=[[-131.974796875,268.0959375,19.5],[0.155328259148464,-0.159070324816329,0.69756522559825,-0.681155283110099],[0,0,0,0],[8.999999E+09,8.999999E+09,8.999999E+09,8.999999E+09,8.999999E+09,8.999999E+09]];
	LOCAL CONST Robtarget Tr_meulage_bavure_P22 :=[[-133.775234375,266.8183125,19.5],[0.158904909325867,-0.16277995359473,0.696812045885557,-0.680224146299306],[0,0,0,0],[8.999999E+09,8.999999E+09,8.999999E+09,8.999999E+09,8.999999E+09,8.999999E+09]];
	LOCAL CONST Robtarget Tr_meulage_bavure_P23 :=[[-134.549140625,266.27978125,19.5],[0.161247588459805,-0.16522852975596,0.696341430548334,-0.679564095779406],[0,0,0,0],[8.999999E+09,8.999999E+09,8.999999E+09,8.999999E+09,8.999999E+09,8.999999E+09]];
	LOCAL CONST Robtarget Tr_meulage_bavure_P24 :=[[-135.5440625,265.107,19.5],[0.162353499588889,-0.166411711557204,0.696167409168838,-0.679190269246395],[0,0,0,0],[8.999999E+09,8.999999E+09,8.999999E+09,8.999999E+09,8.999999E+09,8.999999E+09]];
	LOCAL CONST Robtarget Tr_meulage_bavure_P25 :=[[-138.35925,262.71625,19.5],[0.162258149983295,-0.166365545965166,0.696289691871871,-0.679099008151747],[0,0,0,0],[8.999999E+09,8.999999E+09,8.999999E+09,8.999999E+09,8.999999E+09,8.999999E+09]];
	LOCAL CONST Robtarget Tr_meulage_bavure_P26 :=[[-140.566046875,261.220953125,19.5],[0.161033401452568,-0.165161967639623,0.696689475762883,-0.679274276285554],[0,0,0,0],[8.999999E+09,8.999999E+09,8.999999E+09,8.999999E+09,8.999999E+09,8.999999E+09]];
	LOCAL CONST Robtarget Tr_meulage_bavure_P27 :=[[-141.371765625,260.694578125,19.5],[0.158804492280744,-0.162927378820907,0.697328639470657,-0.679682698791139],[0,0,0,0],[8.999999E+09,8.999999E+09,8.999999E+09,8.999999E+09,8.999999E+09,8.999999E+09]];
	LOCAL CONST Robtarget Tr_meulage_bavure_P28 :=[[-143.899296875,259.55840625,19.5],[0.155733726825713,-0.159828247727153,0.69816049554749,-0.680274841526809],[0,0,0,0],[8.999999E+09,8.999999E+09,8.999999E+09,8.999999E+09,8.999999E+09,8.999999E+09]];
	LOCAL CONST Robtarget Tr_meulage_bavure_P29 :=[[-145.116140625,259.16540625,19.5],[0.151985546193605,-0.156034804423043,0.699140144751935,-0.680996763247182],[0,0,0,0],[8.999999E+09,8.999999E+09,8.999999E+09,8.999999E+09,8.999999E+09,8.999999E+09]];
	LOCAL CONST Robtarget Tr_meulage_bavure_P30 :=[[-148.73684375,258.320671875,19.5],[0.147757614271946,-0.151748975705773,0.700211638166787,-0.681794395380819],[0,0,0,0],[8.999999E+09,8.999999E+09,8.999999E+09,8.999999E+09,8.999999E+09,8.999999E+09]];
	LOCAL CONST Robtarget Tr_meulage_bavure_P31 :=[[-148.770484375,258.310796875,19.5],[0.143236343515947,-0.147157853723554,0.701317472183737,-0.682628536755879],[0,0,0,0],[8.999999E+09,8.999999E+09,8.999999E+09,8.999999E+09,8.999999E+09,8.999999E+09]];
	LOCAL CONST Robtarget Tr_meulage_bavure_P32 :=[[-148.892671875,258.275328125,19.5],[0.138598015602648,-0.142445266090557,0.702421494370918,-0.683450057052543],[0,0,0,0],[8.999999E+09,8.999999E+09,8.999999E+09,8.999999E+09,8.999999E+09,8.999999E+09]];
	LOCAL CONST Robtarget Tr_meulage_bavure_P33 :=[[-151.44721875,257.3569375,19.5],[0.133990268102373,-0.137758644779337,0.7034820656238,-0.68423837015187],[0,0,0,0],[8.999999E+09,8.999999E+09,8.999999E+09,8.999999E+09,8.999999E+09,8.999999E+09]];
	LOCAL CONST Robtarget Tr_meulage_bavure_P34 :=[[-151.79003125,257.2784375,19.5],[0.129554630124136,-0.13324637933274,0.704478763892463,-0.68496034296349],[0,0,0,0],[8.999999E+09,8.999999E+09,8.999999E+09,8.999999E+09,8.999999E+09,8.999999E+09]];
	LOCAL CONST Robtarget Tr_meulage_bavure_P35 :=[[-157.227421875,255.522640625,19.5],[0.125382137768249,-0.129003157908596,0.705400378631081,-0.68560032862113],[0,0,0,0],[8.999999E+09,8.999999E+09,8.999999E+09,8.999999E+09,8.999999E+09,8.999999E+09]];
	LOCAL CONST Robtarget Tr_meulage_bavure_P36 :=[[-158.71228125,255.282109375,19.5],[0.121558679414207,-0.125116371375017,0.706233303859003,-0.686151515041262],[0,0,0,0],[8.999999E+09,8.999999E+09,8.999999E+09,8.999999E+09,8.999999E+09,8.999999E+09]];
	LOCAL CONST Robtarget Tr_meulage_bavure_P37 :=[[-166.161109375,253.328859375,19.5],[0.11811544483246,-0.12162037955801,0.706983271642525,-0.68660897065639],[0,0,0,0],[8.999999E+09,8.999999E+09,8.999999E+09,8.999999E+09,8.999999E+09,8.999999E+09]];
	LOCAL CONST Robtarget Tr_meulage_bavure_P38 :=[[-167.27478125,252.952453125,19.5],[0.115075912252495,-0.11853727354559,0.707645601771974,-0.686981914967501],[0,0,0,0],[8.999999E+09,8.999999E+09,8.999999E+09,8.999999E+09,8.999999E+09,8.999999E+09]];
	LOCAL CONST Robtarget Tr_meulage_bavure_P39 :=[[-167.68021875,252.836859375,19.5],[0.112433531664999,-0.115862133011752,0.708230774168753,-0.687272753433185],[0,0,0,0],[8.999999E+09,8.999999E+09,8.999999E+09,8.999999E+09,8.999999E+09,8.999999E+09]];
	LOCAL CONST Robtarget Tr_meulage_bavure_P40 :=[[-170.5921875,251.858453125,19.5],[0.110178204059138,-0.113581468469378,0.708734925934783,-0.687498958639836],[0,0,0,0],[8.999999E+09,8.999999E+09,8.999999E+09,8.999999E+09,8.999999E+09,8.999999E+09]];
	LOCAL CONST Robtarget Tr_meulage_bavure_P41 :=[[-173.194046875,250.98975,19.5],[0.108275378069529,-0.111665273345408,0.709182613278229,-0.687653495778549],[0,0,0,0],[8.999999E+09,8.999999E+09,8.999999E+09,8.999999E+09,8.999999E+09,8.999999E+09]];
	LOCAL CONST Robtarget Tr_meulage_bavure_P42 :=[[-174.642265625,250.80840625,19.5],[0.106699491429244,-0.110082594687597,0.709566086983139,-0.687759412206786],[0,0,0,0],[8.999999E+09,8.999999E+09,8.999999E+09,8.999999E+09,8.999999E+09,8.999999E+09]];
	LOCAL CONST Robtarget Tr_meulage_bavure_P43 :=[[-176.47209375,250.262078125,19.5],[0.105400651794574,-0.10878500299433,0.709903441435399,-0.687818020673332],[0,0,0,0],[8.999999E+09,8.999999E+09,8.999999E+09,8.999999E+09,8.999999E+09,8.999999E+09]];
	LOCAL CONST Robtarget Tr_meulage_bavure_P44 :=[[-179.45028125,249.50646875,19.5],[0.104347699792812,-0.107743102207047,0.710208782063385,-0.687827352869014],[0,0,0,0],[8.999999E+09,8.999999E+09,8.999999E+09,8.999999E+09,8.999999E+09,8.999999E+09]];
	LOCAL CONST Robtarget Tr_meulage_bavure_P45 :=[[-179.990484375,249.348578125,19.5],[0.10349942093044,-0.106909657555274,0.71047429110726,-0.687811367065211],[0,0,0,0],[8.999999E+09,8.999999E+09,8.999999E+09,8.999999E+09,8.999999E+09,8.999999E+09]];
	LOCAL CONST Robtarget Tr_meulage_bavure_P46 :=[[-182.07434375,248.8176875,19.5],[0.102816921271874,-0.106247801484268,0.710716257829388,-0.687766302051012],[0,0,0,0],[8.999999E+09,8.999999E+09,8.999999E+09,8.999999E+09,8.999999E+09,8.999999E+09]];
	LOCAL CONST Robtarget Tr_meulage_bavure_P47 :=[[-183.2953125,248.44921875,19.5],[0.102273679194688,-0.105730060700632,0.710938455307536,-0.687697434612895],[0,0,0,0],[8.999999E+09,8.999999E+09,8.999999E+09,8.999999E+09,8.999999E+09,8.999999E+09]];
	LOCAL CONST Robtarget Tr_meulage_bavure_P48 :=[[-189.02165625,246.421453125,19.5],[0.101842227614736,-0.105325393142779,0.711136472051906,-0.687618819078824],[0,0,0,0],[8.999999E+09,8.999999E+09,8.999999E+09,8.999999E+09,8.999999E+09,8.999999E+09]];
	LOCAL CONST Robtarget Tr_meulage_bavure_P49 :=[[-190.247734375,246.2606875,19.5],[0.101503889776433,-0.105018670589077,0.711326241517786,-0.687519466863402],[0,0,0,0],[8.999999E+09,8.999999E+09,8.999999E+09,8.999999E+09,8.999999E+09,8.999999E+09]];
	LOCAL CONST Robtarget Tr_meulage_bavure_P50 :=[[-192.2918125,245.6845625,19.5],[0.101240605785992,-0.104788611296794,0.711502021589216,-0.687411492453417],[0,0,0,0],[8.999999E+09,8.999999E+09,8.999999E+09,8.999999E+09,8.999999E+09,8.999999E+09]];
	LOCAL CONST Robtarget Tr_meulage_bavure_P51 :=[[-195.15565625,244.955875,19.5],[0.101029671065717,-0.104612150924158,0.71166844924112,-0.687297113189131],[0,0,0,0],[8.999999E+09,8.999999E+09,8.999999E+09,8.999999E+09,8.999999E+09,8.999999E+09]];
	LOCAL CONST Robtarget Tr_meulage_bavure_P52 :=[[-195.787359375,244.768671875,19.5],[0.100870494387268,-0.104488832764386,0.711825935786674,-0.687176152329975],[0,0,0,0],[8.999999E+09,8.999999E+09,8.999999E+09,8.999999E+09,8.999999E+09,8.999999E+09]];
	LOCAL CONST Robtarget Tr_meulage_bavure_P53 :=[[-197.894859375,244.14484375,19.5],[0.100758207771371,-0.104414827795635,0.711978940941353,-0.687045351457338],[0,0,0,0],[8.999999E+09,8.999999E+09,8.999999E+09,8.999999E+09,8.999999E+09,8.999999E+09]];
	LOCAL CONST Robtarget Tr_meulage_bavure_P54 :=[[-198.898515625,243.783515625,19.5],[0.100689154585056,-0.104383898483252,0.712119987052904,-0.686913982916462],[0,0,0,0],[8.999999E+09,8.999999E+09,8.999999E+09,8.999999E+09,8.999999E+09,8.999999E+09]];
	LOCAL CONST Robtarget Tr_meulage_bavure_P55 :=[[-199.062046875,243.742984375,19.5],[0.100659383389278,-0.104392164332079,0.712250205638381,-0.686782068148141],[0,0,0,0],[8.999999E+09,8.999999E+09,8.999999E+09,8.999999E+09,8.999999E+09,8.999999E+09]];
	LOCAL CONST Robtarget Tr_meulage_bavure_P56 :=[[-204.744671875,241.8045,19.5],[0.100676763016664,-0.104450658180785,0.712377458984246,-0.686638627900613],[0,0,0,0],[8.999999E+09,8.999999E+09,8.999999E+09,8.999999E+09,8.999999E+09,8.999999E+09]];
	LOCAL CONST Robtarget Tr_meulage_bavure_P57 :=[[-207.207515625,241.0571875,19.5],[0.100732334940695,-0.104545866386655,0.712489392241968,-0.686499835733069],[0,0,0,0],[8.999999E+09,8.999999E+09,8.999999E+09,8.999999E+09,8.999999E+09,8.999999E+09]];
	LOCAL CONST Robtarget Tr_meulage_bavure_P58 :=[[-210.40721875,240.530390625,19.5],[0.100830105268326,-0.104685639855053,0.712597084314346,-0.68635238916056],[0,0,0,0],[8.999999E+09,8.999999E+09,8.999999E+09,8.999999E+09,8.999999E+09,8.999999E+09]];
	LOCAL CONST Robtarget Tr_meulage_bavure_P59 :=[[-214.539296875,239.3644375,19.5],[0.100969005885497,-0.104868522702932,0.712699397376542,-0.686197800765722],[0,0,0,0],[8.999999E+09,8.999999E+09,8.999999E+09,8.999999E+09,8.999999E+09,8.999999E+09]];
	LOCAL CONST Robtarget Tr_meulage_bavure_P60 :=[[-214.61996875,239.34234375,19.5],[0.101156775706281,-0.105100267685052,0.712787665052986,-0.686042990642388],[0,0,0,0],[8.999999E+09,8.999999E+09,8.999999E+09,8.999999E+09,8.999999E+09,8.999999E+09]];
	LOCAL CONST Robtarget Tr_meulage_bavure_P61 :=[[-214.712890625,239.315859375,19.5],[0.101397797873345,-0.105386347819318,0.712863952610958,-0.685884239028441],[0,0,0,0],[8.999999E+09,8.999999E+09,8.999999E+09,8.999999E+09,8.999999E+09,8.999999E+09]];
	LOCAL CONST Robtarget Tr_meulage_bavure_P62 :=[[-219.14228125,237.832640625,19.5],[0.101693743509649,-0.105730624286395,0.712934504133883,-0.685714087965515],[0,0,0,0],[8.999999E+09,8.999999E+09,8.999999E+09,8.999999E+09,8.999999E+09,8.999999E+09]];
	LOCAL CONST Robtarget Tr_meulage_bavure_P63 :=[[-219.7968125,237.729125,19.5],[0.102056457123123,-0.106143113508668,0.712989925072344,-0.685538828775946],[0,0,0,0],[8.999999E+09,8.999999E+09,8.999999E+09,8.999999E+09,8.999999E+09,8.999999E+09]];
	LOCAL CONST Robtarget Tr_meulage_bavure_P64 :=[[-223.453984375,236.61040625,19.5],[0.102509330414114,-0.106650041936764,0.713032210768267,-0.685348577105004],[0,0,0,0],[8.999999E+09,8.999999E+09,8.999999E+09,8.999999E+09,8.999999E+09,8.999999E+09]];
	LOCAL CONST Robtarget Tr_meulage_bavure_P65 :=[[-225.453625,236.2213125,19.5],[0.103067273174069,-0.107264675421936,0.713051491947977,-0.685148886328988],[0,0,0,0],[8.999999E+09,8.999999E+09,8.999999E+09,8.999999E+09,8.999999E+09,8.999999E+09]];
	LOCAL CONST Robtarget Tr_meulage_bavure_P66 :=[[-226.42425,235.934453125,19.5],[0.103778137875918,-0.108037056952373,0.713040417684752,-0.684931715700208],[0,0,0,0],[8.999999E+09,8.999999E+09,8.999999E+09,8.999999E+09,8.999999E+09,8.999999E+09]];
	LOCAL CONST Robtarget Tr_meulage_bavure_P67 :=[[-234.28909375,233.7028125,19.5],[0.104688583241208,-0.109015736780408,0.712990596866976,-0.684689914086987],[0,0,0,0],[8.999999E+09,8.999999E+09,8.999999E+09,8.999999E+09,8.999999E+09,8.999999E+09]];
	LOCAL CONST Robtarget Tr_meulage_bavure_P68 :=[[-234.38978125,233.675421875,19.5],[0.105840610079114,-0.110248132471436,0.712905101295668,-0.684404435324067],[0,0,0,0],[8.999999E+09,8.999999E+09,8.999999E+09,8.999999E+09,8.999999E+09,8.999999E+09]];
	LOCAL CONST Robtarget Tr_meulage_bavure_P69 :=[[-234.471390625,233.64940625,19.5],[0.107313983806485,-0.11181299522481,0.712755729195922,-0.68407662836617],[0,0,0,0],[8.999999E+09,8.999999E+09,8.999999E+09,8.999999E+09,8.999999E+09,8.999999E+09]];
	LOCAL CONST Robtarget Tr_meulage_bavure_P70 :=[[-234.690609375,233.58728125,19.5],[0.109174890138464,-0.113783812756771,0.712541968571686,-0.683679771780453],[0,0,0,0],[8.999999E+09,8.999999E+09,8.999999E+09,8.999999E+09,8.999999E+09,8.999999E+09]];
	LOCAL CONST Robtarget Tr_meulage_bavure_P71 :=[[-239.342359375,231.9585625,19.5],[0.111506718354458,-0.116244160624629,0.712235412135731,-0.683208800135318],[0,0,0,0],[8.999999E+09,8.999999E+09,8.999999E+09,8.999999E+09,8.999999E+09,8.999999E+09]];
	LOCAL CONST Robtarget Tr_meulage_bavure_P72 :=[[-241.05609375,231.723265625,19.5],[0.114402182441893,-0.119293532101534,0.711821823792287,-0.682635250352848],[0,0,0,0],[8.999999E+09,8.999999E+09,8.999999E+09,8.999999E+09,8.999999E+09,8.999999E+09]];
	LOCAL CONST Robtarget Tr_meulage_bavure_P73 :=[[-243.429703125,231.046875,19.5],[0.117951401580306,-0.123025889652367,0.711275789036588,-0.68193756992181],[0,0,0,0],[8.999999E+09,8.999999E+09,8.999999E+09,8.999999E+09,8.999999E+09,8.999999E+09]];
	LOCAL CONST Robtarget Tr_meulage_bavure_P74 :=[[-245.614375,230.45709375,19.5],[0.122246114015868,-0.127535321807242,0.71056357553474,-0.681094732341125],[0,0,0,0],[8.999999E+09,8.999999E+09,8.999999E+09,8.999999E+09,8.999999E+09,8.999999E+09]];
	LOCAL CONST Robtarget Tr_meulage_bavure_P75 :=[[-247.715921875,229.86053125,19.5],[0.127383826216461,-0.13292534317687,0.709654438884342,-0.680069695936759],[0,0,0,0],[8.999999E+09,8.999999E+09,8.999999E+09,8.999999E+09,8.999999E+09,8.999999E+09]];
	LOCAL CONST Robtarget Tr_meulage_bavure_P76 :=[[-251.49471875,228.64440625,19.5],[0.133434149308723,-0.13926557870004,0.708505040270779,-0.678838002986355],[0,0,0,0],[8.999999E+09,8.999999E+09,8.999999E+09,8.999999E+09,8.999999E+09,8.999999E+09]];
	LOCAL CONST Robtarget Tr_meulage_bavure_P77 :=[[-251.83371875,228.5833125,19.5],[0.140474202815185,-0.146643801262364,0.707088185414656,-0.677339569154033],[0,0,0,0],[8.999999E+09,8.999999E+09,8.999999E+09,8.999999E+09,8.999999E+09,8.999999E+09]];
	LOCAL CONST Robtarget Tr_meulage_bavure_P78 :=[[-254.43134375,227.758609375,19.5],[0.14857693095733,-0.155131174330336,0.705340347038595,-0.67553993899522],[0,0,0,0],[8.999999E+09,8.999999E+09,8.999999E+09,8.999999E+09,8.999999E+09,8.999999E+09]];
	LOCAL CONST Robtarget Tr_meulage_bavure_P79 :=[[-255.8114375,227.339484375,19.5],[0.157770834680272,-0.164759546460325,0.703215831564924,-0.673387072797608],[0,0,0,0],[8.999999E+09,8.999999E+09,8.999999E+09,8.999999E+09,8.999999E+09,8.999999E+09]];
	LOCAL CONST Robtarget Tr_meulage_bavure_P80 :=[[-257.434203125,226.680359375,19.5],[0.168108910176913,-0.175583762415949,0.700648779186346,-0.670821157179522],[0,0,0,0],[8.999999E+09,8.999999E+09,8.999999E+09,8.999999E+09,8.999999E+09,8.999999E+09]];
	LOCAL CONST Robtarget Tr_meulage_bavure_P81 :=[[-258.876703125,225.929375,19.5],[0.179594801367018,-0.187610093467437,0.697581467899969,-0.667778597885261],[0,0,0,0],[8.999999E+09,8.999999E+09,8.999999E+09,8.999999E+09,8.999999E+09,8.999999E+09]];
	LOCAL CONST Robtarget Tr_meulage_bavure_P82 :=[[-260.03490625,225.27240625,19.5],[0.19222097339903,-0.200829989389977,0.693945145777335,-0.6641976719315],[0,0,0,0],[8.999999E+09,8.999999E+09,8.999999E+09,8.999999E+09,8.999999E+09,8.999999E+09]];
	LOCAL CONST Robtarget Tr_meulage_bavure_P83 :=[[-261.741671875,224.06884375,19.5],[0.205948317219604,-0.215198851847187,0.689669449723072,-0.660023329070072],[0,0,0,0],[8.999999E+09,8.999999E+09,8.999999E+09,8.999999E+09,8.999999E+09,8.999999E+09]];
	LOCAL CONST Robtarget Tr_meulage_bavure_P84 :=[[-262.5081875,223.512453125,19.5],[0.220733190262535,-0.23067379550951,0.684689935099302,-0.655184059295916],[0,0,0,0],[8.999999E+09,8.999999E+09,8.999999E+09,8.999999E+09,8.999999E+09,8.999999E+09]];
	LOCAL CONST Robtarget Tr_meulage_bavure_P85 :=[[-264.4875625,221.74859375,19.5],[0.236496795057254,-0.247173730635575,0.67894713079241,-0.64961927803914],[0,0,0,0],[8.999999E+09,8.999999E+09,8.999999E+09,8.999999E+09,8.999999E+09,8.999999E+09]];
	LOCAL CONST Robtarget Tr_meulage_bavure_P86 :=[[-264.7845,221.43078125,19.5],[0.253137741284196,-0.264587486227869,0.672382433368819,-0.643285791360402],[0,0,0,0],[8.999999E+09,8.999999E+09,8.999999E+09,8.999999E+09,8.999999E+09,8.999999E+09]];
	LOCAL CONST Robtarget Tr_meulage_bavure_P87 :=[[-266.30134375,219.85028125,19.5],[0.270524564003362,-0.282787595139476,0.664968606461892,-0.636132367299567],[0,0,0,0],[8.999999E+09,8.999999E+09,8.999999E+09,8.999999E+09,8.999999E+09,8.999999E+09]];
	LOCAL CONST Robtarget Tr_meulage_bavure_P88 :=[[-266.74840625,219.34478125,19.5],[0.288511543720273,-0.301609658346413,0.65667063241409,-0.628153153026541],[0,0,0,0],[8.999999E+09,8.999999E+09,8.999999E+09,8.999999E+09,8.999999E+09,8.999999E+09]];
	LOCAL CONST Robtarget Tr_meulage_bavure_P89 :=[[-266.905625,219.137140625,19.5],[0.306918950392811,-0.320875516042448,0.647502145199297,-0.619338867710219],[0,0,0,0],[8.999999E+09,8.999999E+09,8.999999E+09,8.999999E+09,8.999999E+09,8.999999E+09]];
	LOCAL CONST Robtarget Tr_meulage_bavure_P90 :=[[-267.0568125,218.931515625,19.5],[0.325566799077425,-0.340387906198695,0.637479790861357,-0.60972276396368],[0,0,0,0],[8.999999E+09,8.999999E+09,8.999999E+09,8.999999E+09,8.999999E+09,8.999999E+09]];
	LOCAL CONST Robtarget Tr_meulage_bavure_P91 :=[[-268.7323125,216.50121875,19.5],[0.344275918423764,-0.359964752143611,0.62665140686161,-0.599339205697431],[0,0,0,0],[8.999999E+09,8.999999E+09,8.999999E+09,8.999999E+09,8.999999E+09,8.999999E+09]];
	LOCAL CONST Robtarget Tr_meulage_bavure_P92 :=[[-269.32665625,215.369265625,19.5],[0.362839677915133,-0.379379509479547,0.615097083756681,-0.588280658760364],[0,0,0,0],[8.999999E+09,8.999999E+09,8.999999E+09,8.999999E+09,8.999999E+09,8.999999E+09]];
	LOCAL CONST Robtarget Tr_meulage_bavure_P93 :=[[-270.63675,212.875359375,19.5],[0.381069958400764,-0.398443167169849,0.602925562322839,-0.576636363436948],[0,0,0,0],[8.999999E+09,8.999999E+09,8.999999E+09,8.999999E+09,8.999999E+09,8.999999E+09]];
	LOCAL CONST Robtarget Tr_meulage_bavure_P94 :=[[-271.8645,209.139859375,19.5],[0.398777004672225,-0.416960005276891,0.590274137485763,-0.564533167457486],[0,0,0,0],[8.999999E+09,8.999999E+09,8.999999E+09,8.999999E+09,8.999999E+09,8.999999E+09]];
	LOCAL CONST Robtarget Tr_meulage_bavure_P95 :=[[-271.86565625,209.135953125,19.5],[0.415785797429814,-0.434739148074722,0.577299843796345,-0.55213126531617],[0,0,0,0],[8.999999E+09,8.999999E+09,8.999999E+09,8.999999E+09,8.999999E+09,8.999999E+09]];
	LOCAL CONST Robtarget Tr_meulage_bavure_P96 :=[[-271.865875,209.134796875,19.5],[0.43195693274044,-0.45163942589146,0.564168606346888,-0.539582079808544],[0,0,0,0],[8.999999E+09,8.999999E+09,8.999999E+09,8.999999E+09,8.999999E+09,8.999999E+09]];
	LOCAL CONST Robtarget Tr_meulage_bavure_P97 :=[[-271.87046875,209.09353125,19.5],[0.447167358382327,-0.467531167244589,0.551059382324554,-0.527057414713392],[0,0,0,0],[8.999999E+09,8.999999E+09,8.999999E+09,8.999999E+09,8.999999E+09,8.999999E+09]];
	LOCAL CONST Robtarget Tr_meulage_bavure_P98 :=[[-272.50703125,202.791109375,19.5],[0.461340473205216,-0.482325755428971,0.538134656276482,-0.51472121109087],[0,0,0,0],[8.999999E+09,8.999999E+09,8.999999E+09,8.999999E+09,8.999999E+09,8.999999E+09]];
	LOCAL CONST Robtarget Tr_meulage_bavure_P99 :=[[-272.4975625,202.657921875,19.5],[0.474401047645067,-0.495953697234708,0.525575952214658,-0.502736008901433],[0,0,0,0],[8.999999E+09,8.999999E+09,8.999999E+09,8.999999E+09,8.999999E+09,8.999999E+09]];
	LOCAL CONST Robtarget Tr_meulage_bavure_P100 :=[[-272.339,199.592125,19.5],[0.486304642379521,-0.508375633057515,0.51354875762644,-0.491253177143758],[0,0,0,0],[8.999999E+09,8.999999E+09,8.999999E+09,8.999999E+09,8.999999E+09,8.999999E+09]];
	LOCAL CONST Robtarget Tr_meulage_bavure_P101 :=[[-272.24275,199.068421875,19.5],[0.497038645063223,-0.519565365624955,0.502194933889742,-0.480421340629452],[0,0,0,0],[8.999999E+09,8.999999E+09,8.999999E+09,8.999999E+09,8.999999E+09,8.999999E+09]];
	LOCAL CONST Robtarget Tr_meulage_bavure_P102 :=[[-270.555125,191.277125,19.5],[0.50662520460159,-0.529546779928466,0.491620573500641,-0.47034064425764],[0,0,0,0],[8.999999E+09,8.999999E+09,8.999999E+09,8.999999E+09,8.999999E+09,8.999999E+09]];
	LOCAL CONST Robtarget Tr_meulage_bavure_P103 :=[[-269.8068125,188.44890625,19.5],[0.515078514957432,-0.53833586136363,0.481935477462382,-0.461114757259222],[0,0,0,0],[8.999999E+09,8.999999E+09,8.999999E+09,8.999999E+09,8.999999E+09,8.999999E+09]];
	LOCAL CONST Robtarget Tr_meulage_bavure_P104 :=[[-269.31125,186.941796875,19.5],[0.522453648758422,-0.545989727445495,0.473194373703913,-0.452796297597459],[0,0,0,0],[8.999999E+09,8.999999E+09,8.999999E+09,8.999999E+09,8.999999E+09,8.999999E+09]];
	LOCAL CONST Robtarget Tr_meulage_bavure_P105 :=[[-268.65690625,184.4749375,19.5],[0.528806295417257,-0.55257088813919,0.465436391224044,-0.44541921964873],[0,0,0,0],[8.999999E+09,8.999999E+09,8.999999E+09,8.999999E+09,8.999999E+09,8.999999E+09]];
	LOCAL CONST Robtarget Tr_meulage_bavure_P106 :=[[-268.393125,183.774328125,19.5],[0.534197117848944,-0.558150922645131,0.458678250363578,-0.438993450379021],[0,0,0,0],[8.999999E+09,8.999999E+09,8.999999E+09,8.999999E+09,8.999999E+09,8.999999E+09]];
	LOCAL CONST Robtarget Tr_meulage_bavure_P107 :=[[-267.63103125,180.726875,19.5],[0.538711598379474,-0.562796668352238,0.452896233510209,-0.433514389075288],[0,0,0,0],[8.999999E+09,8.999999E+09,8.999999E+09,8.999999E+09,8.999999E+09,8.999999E+09]];
	LOCAL CONST Robtarget Tr_meulage_bavure_P108 :=[[-267.58671875,180.61596875,19.5],[0.542418995725176,-0.56660325395578,0.448059389223594,-0.428934924448678],[0,0,0,0],[8.999999E+09,8.999999E+09,8.999999E+09,8.999999E+09,8.999999E+09,8.999999E+09]];
	LOCAL CONST Robtarget Tr_meulage_bavure_P109 :=[[-267.2541875,179.38153125,19.5],[0.545411294093081,-0.569658989564049,0.444098861958182,-0.425195668712682],[0,0,0,0],[8.999999E+09,8.999999E+09,8.999999E+09,8.999999E+09,8.999999E+09,8.999999E+09]];
	LOCAL CONST Robtarget Tr_meulage_bavure_P110 :=[[-266.0195625,175.587796875,19.5],[0.547771871324122,-0.572051492066098,0.440940534589993,-0.422225665215311],[0,0,0,0],[8.999999E+09,8.999999E+09,8.999999E+09,8.999999E+09,8.999999E+09,8.999999E+09]];
	LOCAL CONST Robtarget Tr_meulage_bavure_P111 :=[[-265.641125,174.220703125,19.5],[0.549601357214871,-0.573880654249918,0.438476526040125,-0.419925801704351],[0,0,0,0],[8.999999E+09,8.999999E+09,8.999999E+09,8.999999E+09,8.999999E+09,8.999999E+09]];
	LOCAL CONST Robtarget Tr_meulage_bavure_P112 :=[[-265.016,172.483890625,19.5],[0.55097146639003,-0.575233136609742,0.43662307215647,-0.418207573617198],[0,0,0,0],[8.999999E+09,8.999999E+09,8.999999E+09,8.999999E+09,8.999999E+09,8.999999E+09]];
	LOCAL CONST Robtarget Tr_meulage_bavure_P113 :=[[-264.0065,169.331328125,19.5],[0.551975417843148,-0.57619158084371,0.435268225893417,-0.416974785555801],[0,0,0,0],[8.999999E+09,8.999999E+09,8.999999E+09,8.999999E+09,8.999999E+09,8.999999E+09]];
	LOCAL CONST Robtarget Tr_meulage_bavure_P114 :=[[-263.4459375,168.03003125,19.5],[0.552689425805394,-0.576848447980521,0.434309222532909,-0.416119893646324],[0,0,0,0],[8.999999E+09,8.999999E+09,8.999999E+09,8.999999E+09,8.999999E+09,8.999999E+09]];
	LOCAL CONST Robtarget Tr_meulage_bavure_P115 :=[[-262.75525,165.1885,19.5],[0.553183537558501,-0.577280636958644,0.433651352671631,-0.415549689318797],[0,0,0,0],[8.999999E+09,8.999999E+09,8.999999E+09,8.999999E+09,8.999999E+09,8.999999E+09]];
	LOCAL CONST Robtarget Tr_meulage_bavure_P116 :=[[-262.6401875,164.857109375,19.5],[0.553532688073339,-0.577546507396827,0.433198981361894,-0.415186991095635],[0,0,0,0],[8.999999E+09,8.999999E+09,8.999999E+09,8.999999E+09,8.999999E+09,8.999999E+09]];
	LOCAL CONST Robtarget Tr_meulage_bavure_P117 :=[[-262.5576875,164.628328125,19.5],[0.553785566535089,-0.577707679683862,0.432881582096019,-0.414956526655198],[0,0,0,0],[8.999999E+09,8.999999E+09,8.999999E+09,8.999999E+09,8.999999E+09,8.999999E+09]];
	LOCAL CONST Robtarget Tr_meulage_bavure_P118 :=[[-261.8724375,161.280609375,19.5],[0.553984582966436,-0.577820216602442,0.432636459413555,-0.414789793880122],[0,0,0,0],[8.999999E+09,8.999999E+09,8.999999E+09,8.999999E+09,8.999999E+09,8.999999E+09]];
	LOCAL CONST Robtarget Tr_meulage_bavure_P119 :=[[-261.167484375,158.46734375,19.5],[0.5541617986497,-0.577895267671238,0.432426588169554,-0.414667344222518],[0,0,0,0],[8.999999E+09,8.999999E+09,8.999999E+09,8.999999E+09,8.999999E+09,8.999999E+09]];
	LOCAL CONST Robtarget Tr_meulage_bavure_P120 :=[[-260.620734375,156.34915625,19.5],[0.554340656809962,-0.577973516988804,0.432213857053996,-0.414540989092274],[0,0,0,0],[8.999999E+09,8.999999E+09,8.999999E+09,8.999999E+09,8.999999E+09,8.999999E+09]];
	LOCAL CONST Robtarget Tr_meulage_bavure_P121 :=[[-260.040796875,153.905125,19.5],[0.554515447661914,-0.578052398700157,0.432005078045522,-0.414414834681608],[0,0,0,0],[8.999999E+09,8.999999E+09,8.999999E+09,8.999999E+09,8.999999E+09,8.999999E+09]];
	LOCAL CONST Robtarget Tr_meulage_bavure_P122 :=[[-259.574375,152.208375,19.5],[0.554694883950185,-0.578135566873447,0.431789934460209,-0.41428287984692],[0,0,0,0],[8.999999E+09,8.999999E+09,8.999999E+09,8.999999E+09,8.999999E+09,8.999999E+09]];
	LOCAL CONST Robtarget Tr_meulage_bavure_P123 :=[[-258.18903125,146.520390625,19.5],[0.554873475312671,-0.578225772762776,0.431573204626173,-0.41414363589946],[0,0,0,0],[8.999999E+09,8.999999E+09,8.999999E+09,8.999999E+09,8.999999E+09,8.999999E+09]];
	LOCAL CONST Robtarget Tr_meulage_bavure_P124 :=[[-258.167421875,146.4439375,19.5],[0.555036822311294,-0.578296467076994,0.431378919446249,-0.414028440933995],[0,0,0,0],[8.999999E+09,8.999999E+09,8.999999E+09,8.999999E+09,8.999999E+09,8.999999E+09]];
	LOCAL CONST Robtarget Tr_meulage_bavure_P125 :=[[-258.03546875,146.0284375,19.5],[0.555174084692982,-0.578344695025143,0.43121941901957,-0.413943187022094],[0,0,0,0],[8.999999E+09,8.999999E+09,8.999999E+09,8.999999E+09,8.999999E+09,8.999999E+09]];
	LOCAL CONST Robtarget Tr_meulage_bavure_P126 :=[[-256.713921875,142.12771875,19.5],[0.5552803613817,-0.578348404816006,0.431107355169552,-0.413912178160178],[0,0,0,0],[8.999999E+09,8.999999E+09,8.999999E+09,8.999999E+09,8.999999E+09,8.999999E+09]];
	LOCAL CONST Robtarget Tr_meulage_bavure_P127 :=[[-255.81475,139.810640625,19.5],[0.555335584674572,-0.578311660717568,0.431062287725531,-0.413936366574709],[0,0,0,0],[8.999999E+09,8.999999E+09,8.999999E+09,8.999999E+09,8.999999E+09,8.999999E+09]];
	LOCAL CONST Robtarget Tr_meulage_bavure_P128 :=[[-254.889359375,137.4325625,19.5],[0.555348494139824,-0.578214368733872,0.43108192462581,-0.414034501107368],[0,0,0,0],[8.999999E+09,8.999999E+09,8.999999E+09,8.999999E+09,8.999999E+09,8.999999E+09]];
	LOCAL CONST Robtarget Tr_meulage_bavure_P129 :=[[-254.039796875,134.547421875,19.5],[0.555314346885237,-0.578079158521701,0.431163447863949,-0.414184190732018],[0,0,0,0],[8.999999E+09,8.999999E+09,8.999999E+09,8.999999E+09,8.999999E+09,8.999999E+09]];
	LOCAL CONST Robtarget Tr_meulage_bavure_P130 :=[[-253.50634375,133.143859375,19.5],[0.555232581292605,-0.57789796665191,0.431310084324772,-0.414393933317679],[0,0,0,0],[8.999999E+09,8.999999E+09,8.999999E+09,8.999999E+09,8.999999E+09,8.999999E+09]];
	LOCAL CONST Robtarget Tr_meulage_bavure_P131 :=[[-252.805375,130.4038984375,19.5],[0.555115383231954,-0.577678762991618,0.431506301489118,-0.414652227611161],[0,0,0,0],[8.999999E+09,8.999999E+09,8.999999E+09,8.999999E+09,8.999999E+09,8.999999E+09]];
	LOCAL CONST Robtarget Tr_meulage_bavure_P132 :=[[-252.61525,129.9812890625,19.5],[0.554971537564535,-0.577439144321827,0.431736885950085,-0.41493841519948],[0,0,0,0],[8.999999E+09,8.999999E+09,8.999999E+09,8.999999E+09,8.999999E+09,8.999999E+09]];
	LOCAL CONST Robtarget Tr_meulage_bavure_P133 :=[[-252.54175,129.7639453125,19.5],[0.554807808042344,-0.577183766423066,0.431993141247751,-0.415245857086901],[0,0,0,0],[8.999999E+09,8.999999E+09,8.999999E+09,8.999999E+09,8.999999E+09,8.999999E+09]];
	LOCAL CONST Robtarget Tr_meulage_bavure_P134 :=[[-251.83321875,126.4728671875,19.5],[0.554641405526864,-0.576914099456278,0.432256581761854,-0.415568623270928],[0,0,0,0],[8.999999E+09,8.999999E+09,8.999999E+09,8.999999E+09,8.999999E+09,8.999999E+09]];
	LOCAL CONST Robtarget Tr_meulage_bavure_P135 :=[[-251.18278125,124.0530703125,19.5],[0.554471880423962,-0.5766501601315,0.43252096448312,-0.415885972259251],[0,0,0,0],[8.999999E+09,8.999999E+09,8.999999E+09,8.999999E+09,8.999999E+09,8.999999E+09]];
	LOCAL CONST Robtarget Tr_meulage_bavure_P136 :=[[-251.07853125,123.62765625,19.5],[0.554319928420668,-0.57640447241615,0.432760626439434,-0.416179698373327],[0,0,0,0],[8.999999E+09,8.999999E+09,8.999999E+09,8.999999E+09,8.999999E+09,8.999999E+09]];
	LOCAL CONST Robtarget Tr_meulage_bavure_P137 :=[[-250.58646875,121.9696328125,19.5],[0.55418178516155,-0.57618483357495,0.432976989853418,-0.41644268850688],[0,0,0,0],[8.999999E+09,8.999999E+09,8.999999E+09,8.999999E+09,8.999999E+09,8.999999E+09]];
	LOCAL CONST Robtarget Tr_meulage_bavure_P138 :=[[-249.0630625,117.2281796875,19.5],[0.55406946916178,-0.576000157649405,0.433154713221132,-0.416662736688755],[0,0,0,0],[8.999999E+09,8.999999E+09,8.999999E+09,8.999999E+09,8.999999E+09,8.999999E+09]];
	LOCAL CONST Robtarget Tr_meulage_bavure_P139 :=[[-248.246328125,114.0941484375,19.5],[0.553992165468603,-0.575855121922693,0.433282817500363,-0.416832771280948],[0,0,0,0],[8.999999E+09,8.999999E+09,8.999999E+09,8.999999E+09,8.999999E+09,8.999999E+09]];
	LOCAL CONST Robtarget Tr_meulage_bavure_P140 :=[[-248.078984375,113.68625,19.5],[0.553962687266658,-0.575754826867772,0.433346403881787,-0.416944378421735],[0,0,0,0],[8.999999E+09,8.999999E+09,8.999999E+09,8.999999E+09,8.999999E+09,8.999999E+09]];
	LOCAL CONST Robtarget Tr_meulage_bavure_P141 :=[[-248.020015625,113.5232578125,19.5],[0.554005363778048,-0.575732101107553,0.433309481459314,-0.416957429406043],[0,0,0,0],[8.999999E+09,8.999999E+09,8.999999E+09,8.999999E+09,8.999999E+09,8.999999E+09]];
	LOCAL CONST Robtarget Tr_meulage_bavure_P142 :=[[-246.64209375,107.830171875,19.5],[0.554125296156896,-0.575793699881216,0.433164539816602,-0.416863590136635],[0,0,0,0],[8.999999E+09,8.999999E+09,8.999999E+09,8.999999E+09,8.999999E+09,8.999999E+09]];
	LOCAL CONST Robtarget Tr_meulage_bavure_P143 :=[[-246.36196875,106.7711484375,19.5],[0.554345354114835,-0.575954230403874,0.432882860019575,-0.416641791413743],[0,0,0,0],[8.999999E+09,8.999999E+09,8.999999E+09,8.999999E+09,8.999999E+09,8.999999E+09]];
	LOCAL CONST Robtarget Tr_meulage_bavure_P144 :=[[-246.319390625,106.630765625,19.5],[0.554688143702265,-0.576258876628296,0.43242563593275,-0.416238921451835],[0,0,0,0],[8.999999E+09,8.999999E+09,8.999999E+09,8.999999E+09,8.999999E+09,8.999999E+09]];
	LOCAL CONST Robtarget Tr_meulage_bavure_P145 :=[[-244.73621875,101.860625,19.5],[0.5551689534056,-0.576713575093983,0.431774113546521,-0.41564407892807],[0,0,0,0],[8.999999E+09,8.999999E+09,8.999999E+09,8.999999E+09,8.999999E+09,8.999999E+09]];
	LOCAL CONST Robtarget Tr_meulage_bavure_P146 :=[[-244.059515625,99.5985703125,19.5],[0.555790182505534,-0.577320884426159,0.430923593032146,-0.41485265625777],[0,0,0,0],[8.999999E+09,8.999999E+09,8.999999E+09,8.999999E+09,8.999999E+09,8.999999E+09]];
	LOCAL CONST Robtarget Tr_meulage_bavure_P147 :=[[-243.450703125,98.1990390625,19.5],[0.556572810343997,-0.578099325790582,0.429844061120253,-0.413838083585729],[0,0,0,0],[8.999999E+09,8.999999E+09,8.999999E+09,8.999999E+09,8.999999E+09,8.999999E+09]];
	LOCAL CONST Robtarget Tr_meulage_bavure_P148 :=[[-242.686140625,95.3983125,19.5],[0.557494832159646,-0.579025744502409,0.428563853997992,-0.41262782548576],[0,0,0,0],[8.999999E+09,8.999999E+09,8.999999E+09,8.999999E+09,8.999999E+09,8.999999E+09]];
	LOCAL CONST Robtarget Tr_meulage_bavure_P149 :=[[-242.53040625,95.0535546875,19.5],[0.558545989633152,-0.580080035745051,0.427097995899909,-0.411243032151336],[0,0,0,0],[8.999999E+09,8.999999E+09,8.999999E+09,8.999999E+09,8.999999E+09,8.999999E+09]];
	LOCAL CONST Robtarget Tr_meulage_bavure_P150 :=[[-242.46225,94.838015625,19.5],[0.559681953592698,-0.581238581732019,0.425498572048065,-0.409717936041212],[0,0,0,0],[8.999999E+09,8.999999E+09,8.999999E+09,8.999999E+09,8.999999E+09,8.999999E+09]];
	LOCAL CONST Robtarget Tr_meulage_bavure_P151 :=[[-241.811375,91.6013828125,19.5],[0.560839075192515,-0.582415844291289,0.423861024766721,-0.408158238602842],[0,0,0,0],[8.999999E+09,8.999999E+09,8.999999E+09,8.999999E+09,8.999999E+09,8.999999E+09]];
	LOCAL CONST Robtarget Tr_meulage_bavure_P152 :=[[-241.115,88.9841015625,19.5],[0.561947903583219,-0.58355036123428,0.422280522825776,-0.40664811520989],[0,0,0,0],[8.999999E+09,8.999999E+09,8.999999E+09,8.999999E+09,8.999999E+09,8.999999E+09]];
	LOCAL CONST Robtarget Tr_meulage_bavure_P153 :=[[-241.040296875,88.65740625,19.5],[0.562939042706481,-0.584565844171207,0.4208597002871,-0.40528942830941],[0,0,0,0],[8.999999E+09,8.999999E+09,8.999999E+09,8.999999E+09,8.999999E+09,8.999999E+09]];
	LOCAL CONST Robtarget Tr_meulage_bavure_P154 :=[[-240.501671875,86.4736953125,19.5],[0.563724547845557,-0.585379072843015,0.419725340789636,-0.404198730246397],[0,0,0,0],[8.999999E+09,8.999999E+09,8.999999E+09,8.999999E+09,8.999999E+09,8.999999E+09]];
	LOCAL CONST Robtarget Tr_meulage_bavure_P155 :=[[-239.337734375,81.9293203125,19.5],[0.564235333680435,-0.585911111141601,0.418983986277735,-0.403483676634088],[0,0,0,0],[8.999999E+09,8.999999E+09,8.999999E+09,8.999999E+09,8.999999E+09,8.999999E+09]];
	LOCAL CONST Robtarget Tr_meulage_bavure_P156 :=[[-237.91334375,76.9110390625,19.5],[0.564405931857272,-0.586103743109401,0.418730224063512,-0.403228652073728],[0,0,0,0],[8.999999E+09,8.999999E+09,8.999999E+09,8.999999E+09,8.999999E+09,8.999999E+09]];
	LOCAL CONST Robtarget Tr_meulage_bavure_P157 :=[[-237.585796875,75.893375,19.5],[0.564226085124321,-0.585922409162815,0.418989442649248,-0.403474537306381],[0,0,0,0],[8.999999E+09,8.999999E+09,8.999999E+09,8.999999E+09,8.999999E+09,8.999999E+09]];
	LOCAL CONST Robtarget Tr_meulage_bavure_P158 :=[[-236.730640625,73.168765625,19.5],[0.563690511607683,-0.585386239107043,0.41975853854231,-0.404201345258034],[0,0,0,0],[8.999999E+09,8.999999E+09,8.999999E+09,8.999999E+09,8.999999E+09,8.999999E+09]];
	LOCAL CONST Robtarget Tr_meulage_bavure_P159 :=[[-236.5973125,72.7695625,19.5],[0.562837284012934,-0.584524163608984,0.420982511950505,-0.405363316685174],[0,0,0,0],[8.999999E+09,8.999999E+09,8.999999E+09,8.999999E+09,8.999999E+09,8.999999E+09]];
	LOCAL CONST Robtarget Tr_meulage_bavure_P160 :=[[-235.642984375,69.996640625,19.5],[0.561731815189119,-0.583411212529989,0.422559085765942,-0.406856908427614],[0,0,0,0],[8.999999E+09,8.999999E+09,8.999999E+09,8.999999E+09,8.999999E+09,8.999999E+09]];
	LOCAL CONST Robtarget Tr_meulage_bavure_P161 :=[[-235.146421875,68.4099765625,19.5],[0.560473080509168,-0.582141106136337,0.424344752785144,-0.408550106296205],[0,0,0,0],[8.999999E+09,8.999999E+09,8.999999E+09,8.999999E+09,8.999999E+09,8.999999E+09]];
	LOCAL CONST Robtarget Tr_meulage_bavure_P162 :=[[-234.1725,65.6403203125,19.5],[0.559143909705147,-0.580798622337793,0.426218755242746,-0.410327456075618],[0,0,0,0],[8.999999E+09,8.999999E+09,8.999999E+09,8.999999E+09,8.999999E+09,8.999999E+09]];
	LOCAL CONST Robtarget Tr_meulage_bavure_P163 :=[[-233.90115625,64.58258203125,19.5],[0.557820119701665,-0.579475613934435,0.428068134850034,-0.41207086628072],[0,0,0,0],[8.999999E+09,8.999999E+09,8.999999E+09,8.999999E+09,8.999999E+09,8.999999E+09]];
	LOCAL CONST Robtarget Tr_meulage_bavure_P164 :=[[-233.31884375,63.19534375,19.5],[0.55657665934059,-0.578232527436169,0.429794678183109,-0.413698079639641],[0,0,0,0],[8.999999E+09,8.999999E+09,8.999999E+09,8.999999E+09,8.999999E+09,8.999999E+09]];
	LOCAL CONST Robtarget Tr_meulage_bavure_P165 :=[[-232.660296875,60.35671875,19.5],[0.555482047555963,-0.577152861257167,0.431301136400225,-0.415106732450311],[0,0,0,0],[8.999999E+09,8.999999E+09,8.999999E+09,8.999999E+09,8.999999E+09,8.999999E+09]];
	LOCAL CONST Robtarget Tr_meulage_bavure_P166 :=[[-232.53584375,60.04083203125,19.5],[0.554572637878181,-0.576261331647559,0.432545031829394,-0.416265374976501],[0,0,0,0],[8.999999E+09,8.999999E+09,8.999999E+09,8.999999E+09,8.999999E+09,8.999999E+09]];
	LOCAL CONST Robtarget Tr_meulage_bavure_P167 :=[[-231.62078125,56.0104375,19.5],[0.553862611112111,-0.575587538214364,0.433505283331219,-0.41714309677654],[0,0,0,0],[8.999999E+09,8.999999E+09,8.999999E+09,8.999999E+09,8.999999E+09,8.999999E+09]];
	LOCAL CONST Robtarget Tr_meulage_bavure_P168 :=[[-230.99446875,53.703796875,19.5],[0.55336663976361,-0.575146284877269,0.434164698520518,-0.417723745491197],[0,0,0,0],[8.999999E+09,8.999999E+09,8.999999E+09,8.999999E+09,8.999999E+09,8.999999E+09]];
	LOCAL CONST Robtarget Tr_meulage_bavure_P169 :=[[-230.2911875,51.3466171875,19.5],[0.553075122414816,-0.574918962082387,0.434541292898039,-0.418031052399756],[0,0,0,0],[8.999999E+09,8.999999E+09,8.999999E+09,8.999999E+09,8.999999E+09,8.999999E+09]];
	LOCAL CONST Robtarget Tr_meulage_bavure_P170 :=[[-229.640890625,49.19415234375,19.5],[0.552972758844466,-0.574894376263557,0.434655569132468,-0.418081475718079],[0,0,0,0],[8.999999E+09,8.999999E+09,8.999999E+09,8.999999E+09,8.999999E+09,8.999999E+09]];
	LOCAL CONST Robtarget Tr_meulage_bavure_P171 :=[[-228.847625,47.24008203125,19.5],[0.553039847614054,-0.575055059663213,0.434533817693877,-0.417898273012879],[0,0,0,0],[8.999999E+09,8.999999E+09,8.999999E+09,8.999999E+09,8.999999E+09,8.999999E+09]];
	LOCAL CONST Robtarget Tr_meulage_bavure_P172 :=[[-228.111859375,44.65576171875,19.5],[0.55323919241411,-0.57535331938716,0.434229740622172,-0.417539801942715],[0,0,0,0],[8.999999E+09,8.999999E+09,8.999999E+09,8.999999E+09,8.999999E+09,8.999999E+09]];
	LOCAL CONST Robtarget Tr_meulage_bavure_P173 :=[[-227.846046875,44.0992421875,19.5],[0.553536227427889,-0.575764362914108,0.433786669672334,-0.417039768532447],[0,0,0,0],[8.999999E+09,8.999999E+09,8.999999E+09,8.999999E+09,8.999999E+09,8.999999E+09]];
	LOCAL CONST Robtarget Tr_meulage_bavure_P174 :=[[-227.086890625,41.091734375,19.5],[0.55391940877036,-0.576254157333394,0.433227030419113,-0.416435799202845],[0,0,0,0],[8.999999E+09,8.999999E+09,8.999999E+09,8.999999E+09,8.999999E+09,8.999999E+09]];
	LOCAL CONST Robtarget Tr_meulage_bavure_P175 :=[[-226.98625,40.77059765625,19.5],[0.554339312231722,-0.57678952966024,0.432612580478938,-0.41577412209051],[0,0,0,0],[8.999999E+09,8.999999E+09,8.999999E+09,8.999999E+09,8.999999E+09,8.999999E+09]];
	LOCAL CONST Robtarget Tr_meulage_bavure_P176 :=[[-226.649015625,39.164640625,19.5],[0.554770997972627,-0.577328513694764,0.431982941856371,-0.415104402564663],[0,0,0,0],[8.999999E+09,8.999999E+09,8.999999E+09,8.999999E+09,8.999999E+09,8.999999E+09]];
	LOCAL CONST Robtarget Tr_meulage_bavure_P177 :=[[-225.75671875,35.85235546875,19.5],[0.55518283485586,-0.577856683939294,0.431375900547464,-0.414449641253263],[0,0,0,0],[8.999999E+09,8.999999E+09,8.999999E+09,8.999999E+09,8.999999E+09,8.999999E+09]];
	LOCAL CONST Robtarget Tr_meulage_bavure_P178 :=[[-225.15271875,33.58776953125,19.5],[0.555551681910757,-0.578341709658451,0.43082672457955,-0.413849645382867],[0,0,0,0],[8.999999E+09,8.999999E+09,8.999999E+09,8.999999E+09,8.999999E+09,8.999999E+09]];
	LOCAL CONST Robtarget Tr_meulage_bavure_P179 :=[[-224.391328125,31.239990234375,19.5],[0.555850219101697,-0.578772684949412,0.430368044993933,-0.413323189440352],[0,0,0,0],[8.999999E+09,8.999999E+09,8.999999E+09,8.999999E+09,8.999999E+09,8.999999E+09]];
	LOCAL CONST Robtarget Tr_meulage_bavure_P180 :=[[-223.58921875,28.07726953125,19.5],[0.556063070997077,-0.579114263388536,0.430028543428412,-0.412911592051],[0,0,0,0],[8.999999E+09,8.999999E+09,8.999999E+09,8.999999E+09,8.999999E+09,8.999999E+09]];
	LOCAL CONST Robtarget Tr_meulage_bavure_P181 :=[[-223.27446875,27.11511328125,19.5],[0.55617214110198,-0.579347012270192,0.429834381425739,-0.412640271156359],[0,0,0,0],[8.999999E+09,8.999999E+09,8.999999E+09,8.999999E+09,8.999999E+09,8.999999E+09]];
	LOCAL CONST Robtarget Tr_meulage_bavure_P182 :=[[-222.07909375,21.902740234375,19.5],[0.556163587183498,-0.579463770895492,0.429802931748876,-0.412520596298938],[0,0,0,0],[8.999999E+09,8.999999E+09,8.999999E+09,8.999999E+09,8.999999E+09,8.999999E+09]];
	LOCAL CONST Robtarget Tr_meulage_bavure_P183 :=[[-221.3590625,19.38885546875,19.5],[0.556036524833302,-0.579448079469917,0.429941018292127,-0.412570026831639],[0,0,0,0],[8.999999E+09,8.999999E+09,8.999999E+09,8.999999E+09,8.999999E+09,8.999999E+09]];
	LOCAL CONST Robtarget Tr_meulage_bavure_P184 :=[[-220.956890625,17.979583984375,19.5],[0.555777714942904,-0.579297352812848,0.430263247111801,-0.412794436471327],[0,0,0,0],[8.999999E+09,8.999999E+09,8.999999E+09,8.999999E+09,8.999999E+09,8.999999E+09]];
	LOCAL CONST Robtarget Tr_meulage_bavure_P185 :=[[-220.140671875,15.81234765625,19.5],[0.555387260324963,-0.579010286200185,0.430769490584604,-0.413194537142727],[0,0,0,0],[8.999999E+09,8.999999E+09,8.999999E+09,8.999999E+09,8.999999E+09,8.999999E+09]];
	LOCAL CONST Robtarget Tr_meulage_bavure_P186 :=[[-219.729390625,14.381927734375,19.5],[0.554875249948081,-0.57860918146649,0.431440785503984,-0.413743544628118],[0,0,0,0],[8.999999E+09,8.999999E+09,8.999999E+09,8.999999E+09,8.999999E+09,8.999999E+09]];
	LOCAL CONST Robtarget Tr_meulage_bavure_P187 :=[[-219.277171875,13.1598203125,19.5],[0.554259972605007,-0.578096599830095,0.432256241031451,-0.41443304178376],[0,0,0,0],[8.999999E+09,8.999999E+09,8.999999E+09,8.999999E+09,8.999999E+09,8.999999E+09]];
	LOCAL CONST Robtarget Tr_meulage_bavure_P188 :=[[-218.256109375,9.4919130859375,19.5],[0.553553524513848,-0.577488244498259,0.433196853595789,-0.415242470129592],[0,0,0,0],[8.999999E+09,8.999999E+09,8.999999E+09,8.999999E+09,8.999999E+09,8.999999E+09]];
	LOCAL CONST Robtarget Tr_meulage_bavure_P189 :=[[-218.04615625,8.8970029296875,19.5],[0.55279047989752,-0.576813861469624,0.434215650204435,-0.416131257740525],[0,0,0,0],[8.999999E+09,8.999999E+09,8.999999E+09,8.999999E+09,8.999999E+09,8.999999E+09]];
	LOCAL CONST Robtarget Tr_meulage_bavure_P190 :=[[-217.94775,8.58935546875,19.5],[0.551998054637366,-0.576111151288568,0.435271144726871,-0.417052897850721],[0,0,0,0],[8.999999E+09,8.999999E+09,8.999999E+09,8.999999E+09,8.999999E+09,8.999999E+09]];
	LOCAL CONST Robtarget Tr_meulage_bavure_P191 :=[[-217.15590625,5.42007421875,19.5],[0.551207804493775,-0.575416345219826,0.436318455118486,-0.417961949993092],[0,0,0,0],[8.999999E+09,8.999999E+09,8.999999E+09,8.999999E+09,8.999999E+09,8.999999E+09]];
	LOCAL CONST Robtarget Tr_meulage_bavure_P192 :=[[-216.061046875,1.6334228515625,19.5],[0.550462740383971,-0.574765066470739,0.43730166110026,-0.418811588918942],[0,0,0,0],[8.999999E+09,8.999999E+09,8.999999E+09,8.999999E+09,8.999999E+09,8.999999E+09]];
	LOCAL CONST Robtarget Tr_meulage_bavure_P193 :=[[-214.97621875,-1.83184814453125,19.5],[0.549802892148149,-0.574196387490743,0.438167437841514,-0.419552839096],[0,0,0,0],[8.999999E+09,8.999999E+09,8.999999E+09,8.999999E+09,8.999999E+09,8.999999E+09]];
	LOCAL CONST Robtarget Tr_meulage_bavure_P194 :=[[-214.144828125,-4.2389833984375,19.5],[0.549258432612163,-0.573753219620687,0.438871923723955,-0.420135515930468],[0,0,0,0],[8.999999E+09,8.999999E+09,8.999999E+09,8.999999E+09,8.999999E+09,8.999999E+09]];
	LOCAL CONST Robtarget Tr_meulage_bavure_P195 :=[[-213.356171875,-7.61346435546875,19.5],[0.548860968851809,-0.573457920479178,0.439376466819225,-0.420530582379219],[0,0,0,0],[8.999999E+09,8.999999E+09,8.999999E+09,8.999999E+09,8.999999E+09,8.999999E+09]];
	LOCAL CONST Robtarget Tr_meulage_bavure_P196 :=[[-213.261875,-7.88363671875,19.5],[0.548631375783423,-0.573340573566424,0.439650905767787,-0.420703317393714],[0,0,0,0],[8.999999E+09,8.999999E+09,8.999999E+09,8.999999E+09,8.999999E+09,8.999999E+09]];
	LOCAL CONST Robtarget Tr_meulage_bavure_P197 :=[[-213.24746875,-7.9585263671875,19.5],[0.548581442569393,-0.573404442525945,0.439682482580219,-0.420648381278342],[0,0,0,0],[8.999999E+09,8.999999E+09,8.999999E+09,8.999999E+09,8.999999E+09,8.999999E+09]];
	LOCAL CONST Robtarget Tr_meulage_bavure_P198 :=[[-213.12475,-8.3936767578125,19.5],[0.548712434006602,-0.573656751549552,0.43946747139761,-0.42035810656101],[0,0,0,0],[8.999999E+09,8.999999E+09,8.999999E+09,8.999999E+09,8.999999E+09,8.999999E+09]];
	LOCAL CONST Robtarget Tr_meulage_bavure_P199 :=[[-210.69165625,-15.90313671875,19.5],[0.549017454797688,-0.574075191828592,0.439019298439093,-0.419856599391364],[0,0,0,0],[8.999999E+09,8.999999E+09,8.999999E+09,8.999999E+09,8.999999E+09,8.999999E+09]];
	LOCAL CONST Robtarget Tr_meulage_bavure_P200 :=[[-209.74103125,-19.6936953125,19.5],[0.549467735673187,-0.574650743929498,0.438369404984774,-0.4191586748819],[0,0,0,0],[8.999999E+09,8.999999E+09,8.999999E+09,8.999999E+09,8.999999E+09,8.999999E+09]];
	LOCAL CONST Robtarget Tr_meulage_bavure_P201 :=[[-208.7415625,-23.2620546875,19.5],[0.550033625937453,-0.575350542018132,0.437557559603859,-0.418303892129938],[0,0,0,0],[8.999999E+09,8.999999E+09,8.999999E+09,8.999999E+09,8.999999E+09,8.999999E+09]];
	LOCAL CONST Robtarget Tr_meulage_bavure_P202 :=[[-207.37159375,-28.88333203125,19.5],[0.550692835126397,-0.576135705451497,0.436618058118253,-0.41733646086749],[0,0,0,0],[8.999999E+09,8.999999E+09,8.999999E+09,8.999999E+09,8.999999E+09,8.999999E+09]];
	LOCAL CONST Robtarget Tr_meulage_bavure_P203 :=[[-207.3414375,-28.96075390625,19.5],[0.551401549654211,-0.576972823940223,0.435606216620011,-0.416300270856721],[0,0,0,0],[8.999999E+09,8.999999E+09,8.999999E+09,8.999999E+09,8.999999E+09,8.999999E+09]];
	LOCAL CONST Robtarget Tr_meulage_bavure_P204 :=[[-207.28575,-29.20199609375,19.5],[0.55212555323761,-0.57782752024736,0.434568340612028,-0.415238591227452],[0,0,0,0],[8.999999E+09,8.999999E+09,8.999999E+09,8.999999E+09,8.999999E+09,8.999999E+09]];
	LOCAL CONST Robtarget Tr_meulage_bavure_P205 :=[[-206.205390625,-32.318298828125,19.5],[0.552837700691719,-0.578656352832001,0.433547166896047,-0.414203037286632],[0,0,0,0],[8.999999E+09,8.999999E+09,8.999999E+09,8.999999E+09,8.999999E+09,8.999999E+09]];
	LOCAL CONST Robtarget Tr_meulage_bavure_P206 :=[[-205.579484375,-33.82296875,19.5],[0.553507261330737,-0.579435851078397,0.432583126216197,-0.413225900751903],[0,0,0,0],[8.999999E+09,8.999999E+09,8.999999E+09,8.999999E+09,8.999999E+09,8.999999E+09]];
	LOCAL CONST Robtarget Tr_meulage_bavure_P207 :=[[-204.490296875,-37.62747265625,19.5],[0.554117167545775,-0.580141585327508,0.431703203302885,-0.412337543600824],[0,0,0,0],[8.999999E+09,8.999999E+09,8.999999E+09,8.999999E+09,8.999999E+09,8.999999E+09]];
	LOCAL CONST Robtarget Tr_meulage_bavure_P208 :=[[-203.820046875,-39.33316015625,19.5],[0.554657694921282,-0.580765220490958,0.43092141464287,-0.411549917427869],[0,0,0,0],[8.999999E+09,8.999999E+09,8.999999E+09,8.999999E+09,8.999999E+09,8.999999E+09]];
	LOCAL CONST Robtarget Tr_meulage_bavure_P209 :=[[-202.492234375,-44.71922265625,19.5],[0.55511321691577,-0.5813126088352,0.430252957345398,-0.410861728456397],[0,0,0,0],[8.999999E+09,8.999999E+09,8.999999E+09,8.999999E+09,8.999999E+09,8.999999E+09]];
	LOCAL CONST Robtarget Tr_meulage_bavure_P210 :=[[-202.40375,-45.0029765625,19.5],[0.555503995346946,-0.58178162479792,0.429678228023552,-0.410270730815169],[0,0,0,0],[8.999999E+09,8.999999E+09,8.999999E+09,8.999999E+09,8.999999E+09,8.999999E+09]];
	LOCAL CONST Robtarget Tr_meulage_bavure_P211 :=[[-202.364703125,-45.15894921875,19.5],[0.555839666029998,-0.582184192604284,0.429183561212003,-0.409762495031867],[0,0,0,0],[8.999999E+09,8.999999E+09,8.999999E+09,8.999999E+09,8.999999E+09,8.999999E+09]];
	LOCAL CONST Robtarget Tr_meulage_bavure_P212 :=[[-201.438453125,-48.19219921875,19.5],[0.556138955556572,-0.58253172627159,0.428745755702536,-0.409320567485374],[0,0,0,0],[8.999999E+09,8.999999E+09,8.999999E+09,8.999999E+09,8.999999E+09,8.999999E+09]];
	LOCAL CONST Robtarget Tr_meulage_bavure_P213 :=[[-200.591765625,-51.32173046875,19.5],[0.556409523993353,-0.582847223708114,0.428348827478686,-0.408919108654594],[0,0,0,0],[8.999999E+09,8.999999E+09,8.999999E+09,8.999999E+09,8.999999E+09,8.999999E+09]];
	LOCAL CONST Robtarget Tr_meulage_bavure_P214 :=[[-199.906796875,-53.70884765625,19.5],[0.556680619048654,-0.583146096990925,0.427956749610399,-0.408534378483329],[0,0,0,0],[8.999999E+09,8.999999E+09,8.999999E+09,8.999999E+09,8.999999E+09,8.999999E+09]];
	LOCAL CONST Robtarget Tr_meulage_bavure_P215 :=[[-199.51653125,-54.86445703125,19.5],[0.556952721802798,-0.583447006947069,0.427562290193449,-0.40814671843039],[0,0,0,0],[8.999999E+09,8.999999E+09,8.999999E+09,8.999999E+09,8.999999E+09,8.999999E+09]];
	LOCAL CONST Robtarget Tr_meulage_bavure_P216 :=[[-198.7994375,-57.5790703125,19.5],[0.557247256990595,-0.583758735643388,0.427139766847232,-0.407741158965075],[0,0,0,0],[8.999999E+09,8.999999E+09,8.999999E+09,8.999999E+09,8.999999E+09,8.999999E+09]];
	LOCAL CONST Robtarget Tr_meulage_bavure_P217 :=[[-198.611109375,-58.0790703125,19.5],[0.557560994075282,-0.584088855296033,0.426689693943193,-0.407310510651786],[0,0,0,0],[8.999999E+09,8.999999E+09,8.999999E+09,8.999999E+09,8.999999E+09,8.999999E+09]];
	LOCAL CONST Robtarget Tr_meulage_bavure_P218 :=[[-198.1878125,-59.48582421875,19.5],[0.557901292592321,-0.584434907518608,0.426205132228858,-0.406855222234292],[0,0,0,0],[8.999999E+09,8.999999E+09,8.999999E+09,8.999999E+09,8.999999E+09,8.999999E+09]];
	LOCAL CONST Robtarget Tr_meulage_bavure_P219 :=[[-196.802203125,-63.25659375,19.5],[0.558258236652534,-0.584794192735858,0.425697359845977,-0.406380672734548],[0,0,0,0],[8.999999E+09,8.999999E+09,8.999999E+09,8.999999E+09,8.999999E+09,8.999999E+09]];
	LOCAL CONST Robtarget Tr_meulage_bavure_P220 :=[[-196.199875,-65.348265625,19.5],[0.55863581963713,-0.585153719293122,0.425166928574288,-0.405899283890086],[0,0,0,0],[8.999999E+09,8.999999E+09,8.999999E+09,8.999999E+09,8.999999E+09,8.999999E+09]];
	LOCAL CONST Robtarget Tr_meulage_bavure_P221 :=[[-195.161703125,-67.876328125,19.5],[0.559009058080455,-0.585503942498214,0.424643635693784,-0.405427908471797],[0,0,0,0],[8.999999E+09,8.999999E+09,8.999999E+09,8.999999E+09,8.999999E+09,8.999999E+09]];
	LOCAL CONST Robtarget Tr_meulage_bavure_P222 :=[[-194.595921875,-70.297359375,19.5],[0.559371411308672,-0.585833055893848,0.424138869765393,-0.404980831628801],[0,0,0,0],[8.999999E+09,8.999999E+09,8.999999E+09,8.999999E+09,8.999999E+09,8.999999E+09]];
	LOCAL CONST Robtarget Tr_meulage_bavure_P223 :=[[-194.32346875,-71.0445859375,19.5],[0.559706991093702,-0.586125895463715,0.423675219514731,-0.404578579705892],[0,0,0,0],[8.999999E+09,8.999999E+09,8.999999E+09,8.999999E+09,8.999999E+09,8.999999E+09]];
	LOCAL CONST Robtarget Tr_meulage_bavure_P224 :=[[-192.991,-77.4168828125,19.5],[0.560004505576051,-0.586367581022645,0.423270441078802,-0.404240209985513],[0,0,0,0],[8.999999E+09,8.999999E+09,8.999999E+09,8.999999E+09,8.999999E+09,8.999999E+09]];
	LOCAL CONST Robtarget Tr_meulage_bavure_P225 :=[[-192.971515625,-77.4912890625,19.5],[0.560255431650247,-0.586546563783147,0.422938166599709,-0.403980552816414],[0,0,0,0],[8.999999E+09,8.999999E+09,8.999999E+09,8.999999E+09,8.999999E+09,8.999999E+09]];
	LOCAL CONST Robtarget Tr_meulage_bavure_P226 :=[[-192.947640625,-77.5875390625,19.5],[0.560456452794655,-0.586648518806325,0.422687600493494,-0.403815889103228],[0,0,0,0],[8.999999E+09,8.999999E+09,8.999999E+09,8.999999E+09,8.999999E+09,8.999999E+09]];
	LOCAL CONST Robtarget Tr_meulage_bavure_P227 :=[[-190.67834375,-84.0751796875,19.5],[0.560591035062738,-0.586677268687515,0.422534880557627,-0.403747134385865],[0,0,0,0],[8.999999E+09,8.999999E+09,8.999999E+09,8.999999E+09,8.999999E+09,8.999999E+09]];
	LOCAL CONST Robtarget Tr_meulage_bavure_P228 :=[[-190.06325,-86.149046875,19.5],[0.560660377428896,-0.586629681984142,0.422480021075521,-0.403777400542055],[0,0,0,0],[8.999999E+09,8.999999E+09,8.999999E+09,8.999999E+09,8.999999E+09,8.999999E+09]];
	LOCAL CONST Robtarget Tr_meulage_bavure_P229 :=[[-189.593609375,-87.2691328125,19.5],[0.560666307011502,-0.586501475602497,0.422522698628114,-0.403910733259458],[0,0,0,0],[8.999999E+09,8.999999E+09,8.999999E+09,8.999999E+09,8.999999E+09,8.999999E+09]];
	LOCAL CONST Robtarget Tr_meulage_bavure_P230 :=[[-189.374640625,-87.8335234375,19.5],[0.560610350247965,-0.58629807082073,0.422659085011021,-0.404140947200837],[0,0,0,0],[8.999999E+09,8.999999E+09,8.999999E+09,8.999999E+09,8.999999E+09,8.999999E+09]];
	LOCAL CONST Robtarget Tr_meulage_bavure_P231 :=[[-188.0455,-93.5737421875,19.5],[0.560496795678376,-0.58601898298292,0.422884590414563,-0.404467201152139],[0,0,0,0],[8.999999E+09,8.999999E+09,8.999999E+09,8.999999E+09,8.999999E+09,8.999999E+09]];
	LOCAL CONST Robtarget Tr_meulage_bavure_P232 :=[[-188.020375,-93.6460859375,19.5],[0.560334247414383,-0.585675017861746,0.423185719717289,-0.404875476232583],[0,0,0,0],[8.999999E+09,8.999999E+09,8.999999E+09,8.999999E+09,8.999999E+09,8.999999E+09]];
	LOCAL CONST Robtarget Tr_meulage_bavure_P233 :=[[-187.95440625,-93.9137890625,19.5],[0.560126568783757,-0.585271263902976,0.42355610961918,-0.405359095859724],[0,0,0,0],[8.999999E+09,8.999999E+09,8.999999E+09,8.999999E+09,8.999999E+09,8.999999E+09]];
	LOCAL CONST Robtarget Tr_meulage_bavure_P234 :=[[-185.1970625,-102.701953125,19.5],[0.559885573481247,-0.584822804720757,0.42397729075951,-0.405898618630746],[0,0,0,0],[8.999999E+09,8.999999E+09,8.999999E+09,8.999999E+09,8.999999E+09,8.999999E+09]];
	LOCAL CONST Robtarget Tr_meulage_bavure_P235 :=[[-184.530296875,-104.640703125,19.5],[0.559623207674558,-0.584330628171634,0.424435994595153,-0.406489445010083],[0,0,0,0],[8.999999E+09,8.999999E+09,8.999999E+09,8.999999E+09,8.999999E+09,8.999999E+09]];
	LOCAL CONST Robtarget Tr_meulage_bavure_P236 :=[[-183.37871875,-109.95259375,19.5],[0.55934905118523,-0.58381996073919,0.42491252450692,-0.407102246245128],[0,0,0,0],[8.999999E+09,8.999999E+09,8.999999E+09,8.999999E+09,8.999999E+09,8.999999E+09]];
	LOCAL CONST Robtarget Tr_meulage_bavure_P237 :=[[-183.205578125,-110.6512109375,19.5],[0.55908119321262,-0.583294302901024,0.42538646209581,-0.407728259340424],[0,0,0,0],[8.999999E+09,8.999999E+09,8.999999E+09,8.999999E+09,8.999999E+09,8.999999E+09]];
	LOCAL CONST Robtarget Tr_meulage_bavure_P238 :=[[-181.14784375,-116.7360859375,19.5],[0.558826239727355,-0.582775678929166,0.425842787764896,-0.408342579153162],[0,0,0,0],[8.999999E+09,8.999999E+09,8.999999E+09,8.999999E+09,8.999999E+09,8.999999E+09]];
	LOCAL CONST Robtarget Tr_meulage_bavure_P239 :=[[-179.967546875,-121.5481875,19.5],[0.558602836442108,-0.58227266256863,0.426258949327831,-0.408931199179035],[0,0,0,0],[8.999999E+09,8.999999E+09,8.999999E+09,8.999999E+09,8.999999E+09,8.999999E+09]];
	LOCAL CONST Robtarget Tr_meulage_bavure_P240 :=[[-179.667765625,-122.4904140625,19.5],[0.558422466791908,-0.581799930104044,0.426617830899413,-0.409475782277354],[0,0,0,0],[8.999999E+09,8.999999E+09,8.999999E+09,8.999999E+09,8.999999E+09,8.999999E+09]];
	LOCAL CONST Robtarget Tr_meulage_bavure_P241 :=[[-179.325296875,-123.576015625,19.5],[0.558295909015858,-0.58137148568671,0.42690343114314,-0.409958941950043],[0,0,0,0],[8.999999E+09,8.999999E+09,8.999999E+09,8.999999E+09,8.999999E+09,8.999999E+09]];
	LOCAL CONST Robtarget Tr_meulage_bavure_P242 :=[[-178.80571875,-126.3882578125,19.5],[0.558231443556811,-0.58099632220127,0.427104232646459,-0.410369228218388],[0,0,0,0],[8.999999E+09,8.999999E+09,8.999999E+09,8.999999E+09,8.999999E+09,8.999999E+09]];
	LOCAL CONST Robtarget Tr_meulage_bavure_P243 :=[[-178.746578125,-126.604765625,19.5],[0.558241281506002,-0.580674102324597,0.427207913221496,-0.410703856072712],[0,0,0,0],[8.999999E+09,8.999999E+09,8.999999E+09,8.999999E+09,8.999999E+09,8.999999E+09]];
	LOCAL CONST Robtarget Tr_meulage_bavure_P244 :=[[-178.510609375,-128.216875,19.5],[0.558320087544627,-0.580416784037586,0.427216128579539,-0.410951841622758],[0,0,0,0],[8.999999E+09,8.999999E+09,8.999999E+09,8.999999E+09,8.999999E+09,8.999999E+09]];
	LOCAL CONST Robtarget Tr_meulage_bavure_P245 :=[[-177.235078125,-132.833109375,19.5],[0.558470119615323,-0.580222108067201,0.427127548474046,-0.411114933007125],[0,0,0,0],[8.999999E+09,8.999999E+09,8.999999E+09,8.999999E+09,8.999999E+09,8.999999E+09]];
	LOCAL CONST Robtarget Tr_meulage_bavure_P246 :=[[-176.80528125,-134.65109375,19.5],[0.558681743375904,-0.580083914718664,0.426954564033904,-0.411202093566836],[0,0,0,0],[8.999999E+09,8.999999E+09,8.999999E+09,8.999999E+09,8.999999E+09,8.999999E+09]];
	LOCAL CONST Robtarget Tr_meulage_bavure_P247 :=[[-176.309671875,-136.351703125,19.5],[0.558948862212768,-0.579983383877348,0.426710217946964,-0.41123452403329],[0,0,0,0],[8.999999E+09,8.999999E+09,8.999999E+09,8.999999E+09,8.999999E+09,8.999999E+09]];
	LOCAL CONST Robtarget Tr_meulage_bavure_P248 :=[[-174.79415625,-141.70721875,19.5],[0.559261722556612,-0.579909760982106,0.426408493929037,-0.411225961128256],[0,0,0,0],[8.999999E+09,8.999999E+09,8.999999E+09,8.999999E+09,8.999999E+09,8.999999E+09]];
	LOCAL CONST Robtarget Tr_meulage_bavure_P249 :=[[-174.539484375,-142.4676875,19.5],[0.559601867011069,-0.579845889399106,0.426074710861213,-0.411199265258608],[0,0,0,0],[8.999999E+09,8.999999E+09,8.999999E+09,8.999999E+09,8.999999E+09,8.999999E+09]];
	LOCAL CONST Robtarget Tr_meulage_bavure_P250 :=[[-173.733828125,-144.984546875,19.5],[0.559948913673255,-0.579774847150729,0.425736126316922,-0.411177688397792],[0,0,0,0],[8.999999E+09,8.999999E+09,8.999999E+09,8.999999E+09,8.999999E+09,8.999999E+09]];
	LOCAL CONST Robtarget Tr_meulage_bavure_P251 :=[[-173.34915625,-146.047421875,19.5],[0.560282615086035,-0.579679458062199,0.425419959147396,-0.41118484346106],[0,0,0,0],[8.999999E+09,8.999999E+09,8.999999E+09,8.999999E+09,8.999999E+09,8.999999E+09]];
	LOCAL CONST Robtarget Tr_meulage_bavure_P252 :=[[-173.14975,-146.75825,19.5],[0.560587478067043,-0.579539499269087,0.425149509521977,-0.411246328584938],[0,0,0,0],[8.999999E+09,8.999999E+09,8.999999E+09,8.999999E+09,8.999999E+09,8.999999E+09]];
	LOCAL CONST Robtarget Tr_meulage_bavure_P253 :=[[-171.7659375,-150.988453125,19.5],[0.560843457293698,-0.579333428070608,0.424953258469884,-0.411390475882266],[0,0,0,0],[8.999999E+09,8.999999E+09,8.999999E+09,8.999999E+09,8.999999E+09,8.999999E+09]];
	LOCAL CONST Robtarget Tr_meulage_bavure_P254 :=[[-170.94540625,-152.8334375,19.5],[0.561039561983913,-0.579052376905786,0.424845669083492,-0.411629824174171],[0,0,0,0],[8.999999E+09,8.999999E+09,8.999999E+09,8.999999E+09,8.999999E+09,8.999999E+09]];
	LOCAL CONST Robtarget Tr_meulage_bavure_P255 :=[[-170.333546875,-155.317859375,19.5],[0.561165201636325,-0.578684161810097,0.424841795150663,-0.411980225782464],[0,0,0,0],[8.999999E+09,8.999999E+09,8.999999E+09,8.999999E+09,8.999999E+09,8.999999E+09]];
	LOCAL CONST Robtarget Tr_meulage_bavure_P256 :=[[-169.90046875,-156.504234375,19.5],[0.561217861398805,-0.578224765523599,0.424945209024436,-0.41244660491912],[0,0,0,0],[8.999999E+09,8.999999E+09,8.999999E+09,8.999999E+09,8.999999E+09,8.999999E+09]];
	LOCAL CONST Robtarget Tr_meulage_bavure_P257 :=[[-168.749,-161.391953125,19.5],[0.561199103724622,-0.57767276881116,0.425154141378827,-0.413029895069548],[0,0,0,0],[8.999999E+09,8.999999E+09,8.999999E+09,8.999999E+09,8.999999E+09,8.999999E+09]];
	LOCAL CONST Robtarget Tr_meulage_bavure_P258 :=[[-168.400109375,-162.513125,19.5],[0.561116159236755,-0.57704203302274,0.42545554943413,-0.41371333483957],[0,0,0,0],[8.999999E+09,8.999999E+09,8.999999E+09,8.999999E+09,8.999999E+09,8.999999E+09]];
	LOCAL CONST Robtarget Tr_meulage_bavure_P259 :=[[-168.314890625,-162.82790625,19.5],[0.560971981933904,-0.576343390049549,0.425841928245232,-0.414484480264006],[0,0,0,0],[8.999999E+09,8.999999E+09,8.999999E+09,8.999999E+09,8.999999E+09,8.999999E+09]];
	LOCAL CONST Robtarget Tr_meulage_bavure_P260 :=[[-167.141765625,-166.017046875,19.5],[0.560791565155131,-0.575588968285748,0.426282363188001,-0.415323376266567],[0,0,0,0],[8.999999E+09,8.999999E+09,8.999999E+09,8.999999E+09,8.999999E+09,8.999999E+09]];
	LOCAL CONST Robtarget Tr_meulage_bavure_P261 :=[[-166.6695625,-167.842890625,19.5],[0.560594436223256,-0.574810794973573,0.426745290725287,-0.416190923616997],[0,0,0,0],[8.999999E+09,8.999999E+09,8.999999E+09,8.999999E+09,8.999999E+09,8.999999E+09]];
	LOCAL CONST Robtarget Tr_meulage_bavure_P262 :=[[-166.07134375,-169.3183125,19.5],[0.560411965070534,-0.574024726354164,0.427192537057148,-0.417061841005008],[0,0,0,0],[8.999999E+09,8.999999E+09,8.999999E+09,8.999999E+09,8.999999E+09,8.999999E+09]];
	LOCAL CONST Robtarget Tr_meulage_bavure_P263 :=[[-165.833171875,-170.0676875,19.5],[0.56026916531472,-0.573270161520189,0.42758530836097,-0.417888248676625],[0,0,0,0],[8.999999E+09,8.999999E+09,8.999999E+09,8.999999E+09,8.999999E+09,8.999999E+09]];
	LOCAL CONST Robtarget Tr_meulage_bavure_P264 :=[[-163.94725,-178.9771875,19.5],[0.560193837217065,-0.572572831501146,0.42788684690992,-0.418635955947727],[0,0,0,0],[8.999999E+09,8.999999E+09,8.999999E+09,8.999999E+09,8.999999E+09,8.999999E+09]];
	LOCAL CONST Robtarget Tr_meulage_bavure_P265 :=[[-163.938484375,-179.00759375,19.5],[0.560203218705077,-0.571956209781279,0.428072440595754,-0.419276082608464],[0,0,0,0],[8.999999E+09,8.999999E+09,8.999999E+09,8.999999E+09,8.999999E+09,8.999999E+09]];
	LOCAL CONST Robtarget Tr_meulage_bavure_P266 :=[[-163.915671875,-179.09871875,19.5],[0.560330986746881,-0.571442330960721,0.428100872774782,-0.419776714941307],[0,0,0,0],[8.999999E+09,8.999999E+09,8.999999E+09,8.999999E+09,8.999999E+09,8.999999E+09]];
	LOCAL CONST Robtarget Tr_meulage_bavure_P267 :=[[-162.475125,-182.650140625,19.5],[0.5605819403188,-0.571048404398246,0.427962547398638,-0.420118633300995],[0,0,0,0],[8.999999E+09,8.999999E+09,8.999999E+09,8.999999E+09,8.999999E+09,8.999999E+09]];
